(* IEC 61131-3 sources: std_i2980_v2.06_cp053/Source/IMM/ieccontrol/ODC1 (part 8) *)

(* ---- ABODC.pu ---- *)
(*
@h    ! WARNING !
@h    The Kemro K2 system (including software) only meets category B according to EN 954-1,
@h    thus it is not intended for usage in safety-relevant control applications in the field
@h    of personal safety (e.g. emergency stop).
@h    To implement potentially necessary safety-relevant control tasks, always use additional
@h    external safety devices that are intended for the particular purpose, and meet the necessary
@h    functional safety.
@h    For further information see EN 954-1 (EN ISO 13849-1) and/or the K2-x00 user manual, chapter
@h    "CE conformity, directives and standards".

*)

IMPORT_OVER_LISTFILE
 SET_ALARM
, START_PROCESS_ALGORITHM
, CHECK_REF
, STOP_PROCESS_ALGORITHM
, FCreateODCVersion
, SET_EVENT
, FGetCatConfigValueString
, cMinMoveIdent
, cCompMold
, cCompEjector
, cMoveBeginSequence
, cMoveEndSequence
, cCompInjection
, cMoveFwd
, cMoveBwd
, cMoveStartParallel
, cMoveEndParallel
, cMoveCooling
, cMoveShake
, cMoveOut
, cMoveNone
, cODCDependencyDontCare
, cCompCore
, cMoveFwdInterPos
, cMaxDeviceMovements
, cMaxODCSteps
, cCompNone
, cMovePlast
, cTimeOutSempahore
, cMaxStartConditions
, cCompOperationMode
, cMoveIncreaseShotCounter
, cMaxMoveDevicesRegistered
, cCycleTimeArraySize
, cAllDevIndex
, cMoveStartCondition
, cMinCompId
, ABInterpreter
, KODC_Builder
, FBGetMoveNumber
, FBAutoManual
, FBDebugTrace
, tsGlbSafetyData
, FBDebugTrace2
, KRTOS_Semaphore
, KODC_Sequence
, tyODCSequenceInternal
, KODC_Movements
, tnOperationMode
, tsStartedMoveDataODCExtended
, tyMovementRegisterList
, tsStartedMoveData
, tsODCDeviceMovementList
, tyODCSequenceBackup
, tnDataState
, tevStopRequest
, tevStartedStopped
, tevStartRequest
, ALARM_EVENT
, tsStartedMoveInfo
, tnODCRecalcMode
, KRTOS_Status
, tyStartCondInstanceData
, tevCheckLocklist
, tsTraceLevel
, tyStartConditionPosArray
, tsDeviceId
, tsActiveSequence
, tyLoopData
, tyODCParallelInfo
, tyStepBwdMovements
, tsSequenceDimension
, tevModifyCycleStartCondition
, tevCycleStart
, tyCycleTime
, ABSequDependencies
, RTC
, KODC_Step
, FBLockUnlock
, FBSetStepState
, tsODCStepPos
, ABODCCheckDependencies
, tMoveIdent
, FBStart
, tevCheckLocklistData
, tevStartRequestData
, tevStopRequestData
, FBStop
, FBCheckPosReached
, tevStartedStoppedData
, tsStartedMoveInfoODCExtended
, ABWaitCycleStart
, KSWO_Status
, ALARM_EVENT_DATA
, tyODCDependencyArray
, TON
, tevModifyCycleStartCondData
, FBAddDependency

END_IMPORT

ALGORITHM_BLOCK ABODC #DUMMY_EDIT_BLOCK

SYSTEM_VAR
 sv_ODCSequence : KODC_Sequence;
 sv_ODCSequenceInt : tyODCSequenceInternal;
 sv_ODCMovements : KODC_Movements;
 sv_dCycleDelaySet : TIME;
 sv_dCycleDelayAct : TIME;
 sv_bFirstCycle : BOOL;
 sv_bInitDone : BOOL;
 sv_bCombinedMovementsInManual : BOOL;
 sv_OperationMode : tnOperationMode;
 sv_StartedManualMovements : tsStartedMoveDataODCExtended;
 sv_MovementsAvailable : tyMovementRegisterList;
 sv_bODCFilesChanged : BOOL;
 sv_bProgramSwitchChanged : BOOL;
 sv_bActivationChanged : BOOL;
 sv_StartedMovements : tsStartedMoveData;
 sv_ODCDeviceMovements : tsODCDeviceMovementList (* list of all devices that registered movements for the ODC *);
 sv_iMovementsAvailable : DINT;
 sv_bAutoCycleRunning : BOOL;
 sv_dMaxCycleTime : TIME;
 sv_dCycleTime : TIME;
 sv_dCycleTimeMachine : TIME (* act. cylce time machine *);
 sv_ODCSequenceGenerateTime : DATE_AND_TIME;
 sv_ODCSequenceBackup : tyODCSequenceBackup;
 sv_iODCSequenceAct : DINT;
 sv_iSequenceToRestore : DINT;
 sv_ODCDescriptionPath : STRING(255);
 sv_DataState : tnDataState;
 sv_iODCSequenceUpdated : DINT;
 sv_iUsedRows : DINT;
 sv_iUsedColumns : DINT;
 sv_iInitOK : DINT (* 0 nothing initialized, 10 sequence array initialized, 20 sequence array + safety initialized *);
 sv_iActiveEditors : DINT;
 sv_StartConditionInstanceData : tyStartCondInstanceData (* list with start condition params for all instances *);
 sv_bUseProgramSwitches : BOOL (* TRUE: create sequence by using program switches; FALSE: use sequence from ODC editor *);
 sv_TraceLevel : tsTraceLevel;
 sv_dCalculatedCycleTime : TIME (* calculated cycle time (written by machine sequencer) *);
 sv_iEditorPropertiesChanged : DINT;
 sv_dAllowedCycleDeviation : TIME;
 sv_dLastCycleTime : TIME;
 sv_bTRUE : BOOL;
 sv_bODCCombinedMoveActive : BOOL (* TRUE: combined movement (for example closing sequence) is active (only in manual mode!) *);
 sv_DeviceId : tsDeviceId;
 sv_bOverrideCoreSafety : BOOL;
 sv_bOverrideEjectorSafety : BOOL;
 sv_ActiveSequence : tsActiveSequence;
 sv_LoopParameter : tyLoopData (* array with data of all programmed loops *);
 sv_InterpreterParallelInfo : tyODCParallelInfo (* internal state information of the interpreter, useful for HMI *);
 sv_bSequenceInterruption : BOOL (* TRUE: sequence is interrupted *);
 di_StepFwd : BOOL;
 di_StepBwd : BOOL;
 sv_bStepBwdActive : BOOL (* TRUE: stepping bwd is active *);
 sv_SequenceDimension : tsSequenceDimension (* contains the maximum size of the sequence array *);
 sv_bRecalcPendingOrActive : BOOL (* The ODC wants to recalc the sequence or a recalc is currently active. Any evStartRequest sent at this time can potentially be ignored if recalculation is already active. *);
END_VAR

SYSTEM_OBJECT
 evStopRequest : tevStopRequest;
 evStartedStopped : tevStartedStopped;
 evStartRequest : tevStartRequest;
 evAlarmFinishCycleAndStop : ALARM_EVENT;
 erODCInitFailed : ALARM;
 erCycleTimeExceeded : ALARM;
 EV_Task_3 : TASK;
 EV_Task_7 : TASK;
 PU_Task_3 : TASK;
 PU_Task_7 : TASK;
 TaskAnalog : TASK;
 TaskMid : TASK;
 erAssert : ALARM;
 TaskSlow : TASK;
 erCompNotInCorrectPosition : ALARM;
 erTeachModeActive : ALARM;
 evCheckLocklist : tevCheckLocklist;
 TaskSequencer : TASK;
 erMovementDuringActiveSequence : ALARM;
 erSequenceDuringActiveMovement : ALARM;
 erMachineSequenceNotCreated : ALARM;
 PU_Task_13 : TASK;
 erNoInverseMovement : ALARM;
 erTooManyStartParallel : ALARM;
 TaskInject : TASK;
 evModifyCycleStartCondition : tevModifyCycleStartCondition;
 evNewCycleStarted : tevCycleStart;
END_OBJECT

VAR_GLOBAL
 MovementsSema : KRTOS_Semaphore (* protects sv_StartedManualMovements *);
END_VAR

VAR_EXTERNAL
 g_SafetyData : tsGlbSafetyData;
 g_iAutoCycleLoopStartLine : DINT;
 g_iAutoCycleLoopEndLine : DINT;
 g_iODCMoveDevicesRegistered : DINT (* number of registered devices with ODC movements  *);
END_VAR

VAR
 abInterpreter : ABInterpreter;
 abKODC_Builder : KODC_Builder;
 fbGetMoveNumber : FBGetMoveNumber;
 fbAutoManual : FBAutoManual;
 fbDebugTrace : FBDebugTrace;
 fbDebugTrace2 : FBDebugTrace2;
 dummy : DINT;
 dummy2 : BOOL;
 mStartedCombinedMovement : tsStartedMoveInfo;
 mRecalcMode : tnODCRecalcMode (* currently active recalc mode, set by aDoPendingRecalc when the ODC decided to start recalculation of the sequence *);
 Status : KRTOS_Status;
 mbStopCycle : BOOL;
 mbStopAfterCycle : BOOL;
 mbCycleTimeRunning : BOOL;
 mbCycleTimeMachineRunning : BOOL (* condition for cycle time machine *);
 mbSequenceChanged : BOOL (* the ODC sequence array possibly changed->need to backup when first started *);
 mbIgnoreProgramSwitchChange : BOOL (* ignore program switch or activation changes during mold data loading *);
 mPendingRecalc : tnODCRecalcMode (* recalculations requested by aSetPendingRecalc but not started yet *);
 mbRecalcActive : BOOL;
 mbEjeBwdAtCycleStart : BOOL (* info if ejector must be bwd at the beginning of the cycle (taken from safety array of first step) *);
 miIndexEjectorInSafetyArray : DINT;
 mStartConditionPosArray : tyStartConditionPosArray (* array with information about the position of each start condition in the internal sequence *);
 mActiveStepBwdMovements : tyStepBwdMovements (* ArrayIndex = column number! *);
 mbResetCycleTime : BOOL;
 mbResetCycleTimeMachine : BOOL;
END_VAR

ALGORITHM aIsAnyColumnActive

VAR_OUTPUT
 bActive : BOOL;
END_VAR

VAR_TEMP
 i : DINT;
END_VAR
#BEGIN_EDIT_BLOCK
(**************************************** WARNING ********************************************
 *** The KEBA Kemro K2 System including software is not intended for safety control tasks! ***
 ***                       For further information see Comment tab!                        ***
 *********************************************************************************************)

bActive := FALSE;
FOR i := 2 TO sv_iUsedColumns DO
   IF sv_InterpreterParallelInfo[i].bColumnActive THEN
      bActive := TRUE;
      EXIT;
   END_IF;
END_FOR;

;#END_EDIT_BLOCK END_ALGORITHM

ALGORITHM aCheckCycleTime

VAR
 CycleTimeArray : tyCycleTime;
 i : DINT := 1;
 dSum : TIME;
 dAverageCycleTime : TIME;
END_VAR
#BEGIN_EDIT_BLOCK
(**************************************** WARNING ********************************************
 *** The KEBA Kemro K2 System including software is not intended for safety control tasks! ***
 ***                       For further information see Comment tab!                        ***
 *********************************************************************************************)

CycleTimeArray[i] := sv_dCycleTime;
dSum := dSum + CycleTimeArray[i];
i := i + 1;

IF i > cCycleTimeArraySize THEN
   //check if cycletime of last x - cycles is stable
   dAverageCycleTime := dSum / cCycleTimeArraySize;

   //-> check deviation between average cycle time and calculated cycle time
   IF (SUB_TIME(dAverageCycleTime, sv_dCalculatedCycleTime)) > sv_dAllowedCycleDeviation THEN
      sv_iEditorPropertiesChanged := sv_iEditorPropertiesChanged + 1;
   END_IF;

   i := 1;
   dSum := t#0s;
END_IF;

;#END_EDIT_BLOCK END_ALGORITHM

(*
Back up the current sequence (sv_ODCSequence)
A backup is only written when sv_ODCSequence is not equal to the last backup
*)

PROCESS_ALGORITHM paBackupSequence ON TaskSlow

#BEGIN_EDIT_BLOCK
(**************************************** WARNING ********************************************
 *** The KEBA Kemro K2 System including software is not intended for safety control tasks! ***
 ***                       For further information see Comment tab!                        ***
 *********************************************************************************************)

IF NOT mbSequenceChanged THEN
   fbDebugTrace2(nODCInterpreter, 'no sequence backup written as sequence did NOT change');
   STOP_PROCESS_ALGORITHM();
   RETURN;
END_IF;

mbSequenceChanged := FALSE;

IF sv_ODCSequenceBackup[sv_iODCSequenceAct].Sequence = sv_ODCSequence THEN
   fbDebugTrace2(nODCInterpreter, 'ODC sequences equal, doing nothing');
   STOP_PROCESS_ALGORITHM();
   RETURN;
END_IF;
fbDebugTrace2(nODCInterpreter, 'ODC sequences different, making backup');

sv_iODCSequenceAct := sv_iODCSequenceAct + 1;
IF sv_iODCSequenceAct > cODCSequenceBackupCount THEN
   sv_iODCSequenceAct := 1;
END_IF;

//FIXME: maybe do in smaller steps to avoid blocking the system for a long time
fbDebugTrace2(nODCInterpreter, CONCAT('saving new ODC sequence in history at pos ', DINT_TO_STRING(sv_iODCSequenceAct)));

sv_ODCSequenceBackup[sv_iODCSequenceAct].Sequence := sv_ODCSequence;
sv_ODCSequenceBackup[sv_iODCSequenceAct].Date := sv_ODCSequenceGenerateTime;
fbDebugTrace2(nODCInterpreter, 'saving backup done');

STOP_PROCESS_ALGORITHM();

;#END_EDIT_BLOCK END_ALGORITHM

(*
Queue a recalculation of the ODC sequence

nODCRecalcReloadFiles reload the ODC files from the CF + nODCRecalcCylce
nODCRecalcCylce       recalculate the cycle(because a program switch changed) + nODCRecalcSafety
nODCRecalcSafety      recalculate safety only(a movement was disabled)
*)

ALGORITHM aSetPendingRecalc

VAR_INPUT
 RecalcMode : tnODCRecalcMode (* How much of the ODC array to recalculate *);
END_VAR
#BEGIN_EDIT_BLOCK
(**************************************** WARNING ********************************************
 *** The KEBA Kemro K2 System including software is not intended for safety control tasks! ***
 ***                       For further information see Comment tab!                        ***
 *********************************************************************************************)

IF RecalcMode > mPendingRecalc THEN
   mPendingRecalc := RecalcMode;
   sv_bRecalcPendingOrActive := TRUE;
END_IF;

;#END_EDIT_BLOCK END_ALGORITHM

(*
Start a pending recalculation of the ODC sequence

If bStartedRecalc is TRUE then a pending recalculation was started.

To find out when recalculation finishes wait until mbRecalcActive is FALSE again
*)

ALGORITHM aDoPendingRecalc

VAR_OUTPUT
 bStartedRecalc : BOOL;
END_VAR
#BEGIN_EDIT_BLOCK
(**************************************** WARNING ********************************************
 *** The KEBA Kemro K2 System including software is not intended for safety control tasks! ***
 ***                       For further information see Comment tab!                        ***
 *********************************************************************************************)

bStartedRecalc := FALSE;

IF mPendingRecalc = nODCRecalcNone THEN
   RETURN;
END_IF;

IF mbRecalcActive THEN
   fbDebugTrace('another ODC recalc is already active, new recalc will be executed later');
   RETURN;
END_IF;

IF mPendingRecalc > mRecalcMode THEN
   mRecalcMode := mPendingRecalc;
END_IF;
// mRecalcMode will be reset after the recalc finished successfully
// but keeps the value if an error occured
// this way we can be sure the right recalc mode is used when
// the first recalc with nODCRecalcCylce fails and the second recalc with only nODCRecalcSafety succeeds
// the cycle is recalculated, and not only safety

mPendingRecalc := nODCRecalcNone;

IF mRecalcMode = nODCRecalcReloadFiles THEN
   fbDebugTrace2(nODCInterpreter, 'start initializing ODC array WITH reading new files');
ELSIF mRecalcMode = nODCRecalcCylce THEN
   fbDebugTrace2(nODCInterpreter, 'start initializing ODC array WITHOUT reading new files');
ELSIF mRecalcMode = nODCRecalcSafety THEN
   fbDebugTrace2(nODCInterpreter, 'start initializing ODC dependency array');
ELSIF mRecalcMode = nODCRecalcInternal THEN
   fbDebugTrace2(nODCInterpreter, 'start initializing internal ODC array');
ELSE
   fbDebugTrace2(nODCInterpreter, 'NOT starting initialization of ODC because we got a strange reason');
   RETURN;
END_IF;

bStartedRecalc := TRUE;
mbRecalcActive := TRUE; //set flag immediately, do not wait for PA, which might be delayed a bit because it is low prio
START_PROCESS_ALGORITHM(paInitSequence);

;#END_EDIT_BLOCK END_ALGORITHM

(*
Does the (re)initialisation of the ODC sequence and saves
the sequence generation time

*)

PROCESS_ALGORITHM paInitSequence ON TaskMid

VAR_TEMP
 iTmpRow : DINT;
 iTmpCol : DINT;
 iMove : DINT;
 iDevice : DINT;
 k : DINT;
 i : DINT;
 iTmpCol2 : DINT (* column *);
 iTmpRow2 : DINT (* line *);
END_VAR

VAR
 iCalledInit : DINT;
 iCalledCreate : DINT;
 bInitDone : BOOL;
 abSequDependencies : ABSequDependencies;
 fbRTC : RTC;
 bError : BOOL;
 RecalcMode : tnODCRecalcMode;
 sPath : STRING(255);
 bFirstCall : BOOL;
 sWorkPath : STRING(255);
 iInstance : DINT;
 fbLockUnlockAll : FBLockUnlock := (DeviceId:=(CompId:=cCompAll,IndexId:=cAllDevIndex),MoveDir:=cMoveAll,MoveId:=cMoveAll);
 DeviceId : tsDeviceId;
 bTryAgain : BOOL;
 FailedRecalc : tnODCRecalcMode;
 iCount : INT;
 iOrigEndLine : DINT;
 StepBeginLoop : KODC_Step := (iCompId:=cCompODC,iMoveDir:=cMoveNone,iMoveId:=cMoveBeginLoop,iIndexId:=1,iCount:=1);
 StepEndLoop : KODC_Step := (iCompId:=cCompODC,iMoveDir:=cMoveNone,iMoveId:=cMoveEndLoop,iIndexId:=1,iCount:=1);
 bAddLoop : BOOL;
 iTmp : DINT;
 DeviceIdEjector1 : tsDeviceId := (CompId:=cCompEjector,IndexId:=1);
 DependencyEjectorBwd : LWORD (* dependency which represents "ejector bwd" *);
 bInit : BOOL;
 iNoOfStartParallel : DINT;
END_VAR

VAR CONSTANT
 EmptySequenceEntry : KODC_Step := (iCompId:=cCompNone,iMoveDir:=cMoveNone,iMoveId:=cMoveNone,iIndexId:=1,iCount:=0);
END_VAR

(* IecGraph-Code *)

(* init step *)
INITIAL_STEP SStart:
AStart (P);
AInitAdditionalMoveData (P);
AResetProgrammedInSequence (P);
END_STEP

ACTION AStart: #BEGIN_EDIT_BLOCK
fbDebugTrace2(nODCInterpreter, 'starting initialisation of ODC sequence');

RESET_ALARM(Name := erODCInitFailed);

RecalcMode := mRecalcMode;
FailedRecalc := mRecalcMode;  //remember in case of failed recalc so we can repeat
mRecalcMode := nODCRecalcNone;

sv_iInitOK := 0;

(* lock all movements so nothing can happen during init *)
fbLockUnlockAll.Alarm.AlarmId := erMachineSequenceNotCreated;
fbLockUnlockAll(Mode := nLockAbort);

;#END_EDIT_BLOCK END_ACTION (*AStart*)

(* steps *)
STEP SError:
AError (N);
END_STEP

ACTION AError: #BEGIN_EDIT_BLOCK
fbDebugTrace('initializing ODC array NOT successful');

(* set the generic erODCInitFailed ALARM which will block machine operation
   for detailed information other alarms are set which explain 1 or more problems
   of the ODC sequence *)
SET_ALARM(Name := erODCInitFailed);

mbRecalcActive := FALSE;

//reset mRecalcMode
//this way a failed recalc can not be replaced by a succeeding recalc
//of lower priority
mRecalcMode := FailedRecalc;

// indicate an update of the odc list so the hmi can react properly
sv_iODCSequenceUpdated := sv_iODCSequenceUpdated + 1;

//notify other code parts when recalc is finished (in this case unsuccessfully)
sv_bRecalcPendingOrActive := FALSE;

STOP_PROCESS_ALGORITHM();

;#END_EDIT_BLOCK END_ACTION (*AError*)
STEP Step28:
END_STEP

STEP SInitSequence:
AInit1 (P);
AInit2 (N);
END_STEP

ACTION AInit1: #BEGIN_EDIT_BLOCK
iCalledInit := 0;
iCalledCreate := 0;

IF NOT bFirstCall THEN
   sWorkPath := FGetCatConfigValueString('System.workPath', '/harddisk0/');
   bFirstCall := TRUE;
END_IF;

sPath := CONCAT(sWorkPath, sv_ODCDescriptionPath);
abKODC_Builder.Init(Movements := sv_ODCMovements, DescriptionFilePath := sPath, Execute := FALSE);

;#END_EDIT_BLOCK END_ACTION (*AInit1*)
ACTION AInit2: #BEGIN_EDIT_BLOCK
abKODC_Builder.Init(Execute := TRUE);
iCalledInit := iCalledInit + 1;

;#END_EDIT_BLOCK END_ACTION (*AInit2*)
STEP SInitSequenceDone:
AInit3 (P);
END_STEP

ACTION AInit3: #BEGIN_EDIT_BLOCK
IF abKODC_Builder.Init.Error AND abKODC_Builder.Init.Done THEN
   fbDebugTrace2(nODCInterpreter, 'ERROR init returned success and failure at the same time');
END_IF;

IF abKODC_Builder.Init.Done THEN
   fbDebugTrace2(nODCInterpreter, CONCAT('called init ',
                                         DINT_TO_STRING(iCalledInit),
                                         ' times then it returned success'));
ELSIF abKODC_Builder.Init.Error THEN
   fbDebugTrace2(nODCInterpreter, CONCAT('called init ',
                                         DINT_TO_STRING(iCalledInit),
                                         ' times then it returned error'));
END_IF;

;#END_EDIT_BLOCK END_ACTION (*AInit3*)
STEP Step16:
END_STEP

STEP SCreateSequence:
AClearSequence (P);
ACreateSequence1 (P);
ACreateSequence2 (N);
END_STEP

ACTION ACreateSequence1: #BEGIN_EDIT_BLOCK
fbDebugTrace2(nODCInterpreter, 'initialisation of ODC array');
(* WARNING: Columns and Rows must be <= the real size of the array
   otherwise the builder will write outside of the array
   and memory corruption will occur ! *)
abKODC_Builder.CreateSequence(Sequence := sv_ODCSequence, Columns := cMaxParallelMovements, Rows := cMaxODCSteps, Execute := FALSE);

;#END_EDIT_BLOCK END_ACTION (*ACreateSequence1*)
ACTION ACreateSequence2: #BEGIN_EDIT_BLOCK
abKODC_Builder.CreateSequence(Execute := TRUE);
iCalledCreate := iCalledCreate + 1;

;#END_EDIT_BLOCK END_ACTION (*ACreateSequence2*)
STEP SCreateSequenceDone:
ACreateSequence3 (P);
END_STEP

ACTION ACreateSequence3: #BEGIN_EDIT_BLOCK
IF abKODC_Builder.CreateSequence.Error AND abKODC_Builder.CreateSequence.Done THEN
   fbDebugTrace2(nODCInterpreter, 'ERROR CreateSequence returned success and failure at the same time');
END_IF;

IF abKODC_Builder.CreateSequence.Done THEN
   fbDebugTrace2(nODCInterpreter, CONCAT('called CreateSequence ',
                                         DINT_TO_STRING(iCalledCreate),
                                         ' times then it returned success'));
ELSIF abKODC_Builder.CreateSequence.Error THEN
   fbDebugTrace2(nODCInterpreter, CONCAT('called CreateSequence ',
                                         DINT_TO_STRING(iCalledCreate),
                                         ' times then it returned error'));
END_IF;

;#END_EDIT_BLOCK END_ACTION (*ACreateSequence3*)
STEP SSanityCheckAndNumber:
ACheckSequenceDimension (P);
AInitEmptySteps (P);
ASanity (P);
END_STEP

ACTION ASanity: #BEGIN_EDIT_BLOCK
bError := FALSE;
abInterpreter.aCheckSequenceSanity();
IF NOT abInterpreter.aCheckSequenceSanity.bOK THEN
   fbDebugTrace('checking sanity of ODC array failed');
   bError := TRUE;
   RETURN;
END_IF;
bAddLoop := NOT abInterpreter.aCheckSequenceSanity.bAutoCycleLoopFound;
iNoOfStartParallel := abInterpreter.aCheckSequenceSanity.iNoOfStartParallel;

;#END_EDIT_BLOCK END_ACTION (*ASanity*)
STEP Step33:
END_STEP

STEP S_AddCycleLoop:
AInsertAutoCycleLoop (P);
END_STEP

STEP Step32:
ACreateInternalSequence (P);
END_STEP

ACTION ACreateInternalSequence: #BEGIN_EDIT_BLOCK
bError := FALSE;
abInterpreter.aClearInternalSequence();

abInterpreter.aCreateInternalSequence();
IF abInterpreter.aCreateInternalSequence.bError THEN
   fbDebugTrace('aCreateInternalSequence failed');
   bError := TRUE;
   RETURN;
END_IF;

sv_iUsedColumns := abInterpreter.aCreateInternalSequence.iUsedColumns;
sv_iUsedRows := abInterpreter.aCreateInternalSequence.iUsedRows;

// save sequence generation time
fbRTC(EN := FALSE);
sv_ODCSequenceGenerateTime := fbRTC.CDT;
mbSequenceChanged := TRUE;

;#END_EDIT_BLOCK END_ACTION (*ACreateInternalSequence*)
STEP Step26:
AInitSequenceOK (N);
END_STEP

ACTION AInitSequenceOK: #BEGIN_EDIT_BLOCK
sv_iInitOK := 10;

;#END_EDIT_BLOCK END_ACTION (*AInitSequenceOK*)
STEP SBeforeRecalcSafety:
END_STEP

STEP SRecalcSafety:
ACalcSeqDependencies (P);
ASetProgrammedInSequence (P);
END_STEP

ACTION ACalcSeqDependencies: #BEGIN_EDIT_BLOCK
IF iNoOfStartParallel <= cMaxStartParallel THEN
   RESET_ALARM(Name := erTooManyStartParallel);
   abSequDependencies.aCalc();
   IF abSequDependencies.aCalc.bError THEN
      bError := TRUE;
      fbDebugTrace('sequence dependency calculation returned a error');
   END_IF;
ELSE
   SET_ALARM(Name := erTooManyStartParallel);
END_IF;

;#END_EDIT_BLOCK END_ACTION (*ACalcSeqDependencies*)
STEP S_Check_Pending_Recalc:
ACheckForPendingRecalc (P);
END_STEP

ACTION ACheckForPendingRecalc: #BEGIN_EDIT_BLOCK
bTryAgain := FALSE;
IF mPendingRecalc <> nODCRecalcNone THEN
   //recalc during creation of sequence requested
   //=> ignore result and start again
   mRecalcMode := mPendingRecalc;
   mPendingRecalc := nODCRecalcNone;
   bTryAgain := TRUE;
END_IF;

;#END_EDIT_BLOCK END_ACTION (*ACheckForPendingRecalc*)
STEP SFinish:
ACheckEjeBwdAtCycleStart (P);
AFinish (N);
END_STEP

ACTION AFinish: #BEGIN_EDIT_BLOCK
(* array ok -> unlock all movements *)
fbLockUnlockAll.Alarm.AlarmId := erMachineSequenceNotCreated;
fbLockUnlockAll(Mode := nUnlock);

abInterpreter.aSetInitOK();
fbDebugTrace2(nODCInterpreter, 'initializing ODC array successful');

mbRecalcActive := FALSE;

// indicate an update of the odc list so the hmi can react properly
sv_iInitOK := 20;
sv_iODCSequenceUpdated := sv_iODCSequenceUpdated + 1;

//notify other code parts when recalc is finished (and it is OK to send an evStartRequest)
sv_bRecalcPendingOrActive := FALSE;

STOP_PROCESS_ALGORITHM();

;#END_EDIT_BLOCK END_ACTION (*AFinish*)

(* transitions *)
TRANSITION Trans25 (* Trans25 *) FROM SError TO SStart :=  #BEGIN_EDIT_BLOCK
TRUE
;#END_EDIT_BLOCK
END_TRANSITION

GO_ON_TRANSITION Trans38 (* Trans38 *) FROM SStart TO Step28 :=  #BEGIN_EDIT_BLOCK
RecalcMode <> nODCRecalcInternal
;#END_EDIT_BLOCK
END_TRANSITION

GO_ON_TRANSITION TNewSequenceFromEditor (* Trans39 *) FROM SStart TO SSanityCheckAndNumber :=  #BEGIN_EDIT_BLOCK
RecalcMode = nODCRecalcInternal
;#END_EDIT_BLOCK
END_TRANSITION

GO_ON_TRANSITION Trans13 (* Trans13 *) FROM Step28 TO Step16 :=  #BEGIN_EDIT_BLOCK
NOT (RecalcMode >= nODCRecalcReloadFiles)
;#END_EDIT_BLOCK
END_TRANSITION

GO_ON_TRANSITION TRecalcReloadFiles (* Trans12 *) FROM Step28 TO SInitSequence :=  #BEGIN_EDIT_BLOCK
RecalcMode >= nODCRecalcReloadFiles
;#END_EDIT_BLOCK
END_TRANSITION

TRANSITION Trans2 (* Trans2 *) FROM SInitSequence TO SInitSequenceDone :=  #BEGIN_EDIT_BLOCK
abKODC_Builder.Init.Done OR abKODC_Builder.Init.Error
;#END_EDIT_BLOCK
END_TRANSITION

GO_ON_TRANSITION Trans11 (* Trans11 *) FROM SInitSequenceDone TO Step16 :=  #BEGIN_EDIT_BLOCK
NOT abKODC_Builder.Init.Error
;#END_EDIT_BLOCK
END_TRANSITION

GO_ON_TRANSITION Trans26 (* Trans26 *) FROM SInitSequenceDone TO SError :=  #BEGIN_EDIT_BLOCK
abKODC_Builder.Init.Error
;#END_EDIT_BLOCK
END_TRANSITION

GO_ON_TRANSITION Trans20 (* Trans20 *) FROM Step16 TO SBeforeRecalcSafety :=  #BEGIN_EDIT_BLOCK
NOT (RecalcMode >= nODCRecalcCylce)
;#END_EDIT_BLOCK
END_TRANSITION

GO_ON_TRANSITION TRecalcCycle (* Trans19 *) FROM Step16 TO SCreateSequence :=  #BEGIN_EDIT_BLOCK
RecalcMode >= nODCRecalcCylce
;#END_EDIT_BLOCK
END_TRANSITION

TRANSITION Trans4 (* Trans4 *) FROM SCreateSequence TO SCreateSequenceDone :=  #BEGIN_EDIT_BLOCK
abKODC_Builder.CreateSequence.Error OR abKODC_Builder.CreateSequence.Done
;#END_EDIT_BLOCK
END_TRANSITION

GO_ON_TRANSITION Trans27 (* Trans27 *) FROM SCreateSequenceDone TO SSanityCheckAndNumber :=  #BEGIN_EDIT_BLOCK
NOT abKODC_Builder.CreateSequence.Error
;#END_EDIT_BLOCK
END_TRANSITION

GO_ON_TRANSITION Trans28 (* Trans28 *) FROM SCreateSequenceDone TO SError :=  #BEGIN_EDIT_BLOCK
abKODC_Builder.CreateSequence.Error
;#END_EDIT_BLOCK
END_TRANSITION

GO_ON_TRANSITION Trans46 (* Trans46 *) FROM SSanityCheckAndNumber TO Step33 :=  #BEGIN_EDIT_BLOCK
NOT bError
;#END_EDIT_BLOCK
END_TRANSITION

GO_ON_TRANSITION Trans50 (* Trans50 *) FROM SSanityCheckAndNumber TO SError :=  #BEGIN_EDIT_BLOCK
bError
;#END_EDIT_BLOCK
END_TRANSITION

GO_ON_TRANSITION Trans48 (* Trans48 *) FROM Step33 TO S_AddCycleLoop :=  #BEGIN_EDIT_BLOCK
bAddLoop
;#END_EDIT_BLOCK
END_TRANSITION

TRANSITION TLoopAdded (* Trans50 *) FROM S_AddCycleLoop TO Step32 :=  #BEGIN_EDIT_BLOCK
TRUE
;#END_EDIT_BLOCK
END_TRANSITION

GO_ON_TRANSITION Trans49 (* Trans49 *) FROM Step33 TO Step32 :=  #BEGIN_EDIT_BLOCK
NOT bAddLoop
;#END_EDIT_BLOCK
END_TRANSITION

TRANSITION Trans14 (* Trans14 *) FROM Step32 TO Step26 :=  #BEGIN_EDIT_BLOCK
NOT bError
;#END_EDIT_BLOCK
END_TRANSITION

GO_ON_TRANSITION Trans36 (* Trans36 *) FROM Step26 TO SBeforeRecalcSafety :=  #BEGIN_EDIT_BLOCK
TRUE
;#END_EDIT_BLOCK
END_TRANSITION

TRANSITION Trans29 (* Trans29 *) FROM Step32 TO SError :=  #BEGIN_EDIT_BLOCK
bError
;#END_EDIT_BLOCK
END_TRANSITION

GO_ON_TRANSITION Trans22 (* Trans22 *) FROM SBeforeRecalcSafety TO S_Check_Pending_Recalc :=  #BEGIN_EDIT_BLOCK
NOT (RecalcMode >= nODCRecalcSafety)
;#END_EDIT_BLOCK
END_TRANSITION

GO_ON_TRANSITION TRecalcSafety (* Trans23 *) FROM SBeforeRecalcSafety TO SRecalcSafety :=  #BEGIN_EDIT_BLOCK
RecalcMode >= nODCRecalcSafety
;#END_EDIT_BLOCK
END_TRANSITION

GO_ON_TRANSITION Trans24 (* Trans24 *) FROM SRecalcSafety TO S_Check_Pending_Recalc :=  #BEGIN_EDIT_BLOCK
NOT bError
;#END_EDIT_BLOCK
END_TRANSITION

GO_ON_TRANSITION Trans30 (* Trans30 *) FROM SRecalcSafety TO SError :=  #BEGIN_EDIT_BLOCK
bError
;#END_EDIT_BLOCK
END_TRANSITION

GO_ON_TRANSITION TNoRecalc (* Trans44 *) FROM S_Check_Pending_Recalc TO SFinish :=  #BEGIN_EDIT_BLOCK
NOT bTryAgain
;#END_EDIT_BLOCK
END_TRANSITION

GO_ON_TRANSITION TRecalc (* Trans45 *) FROM S_Check_Pending_Recalc TO SStart :=  #BEGIN_EDIT_BLOCK
bTryAgain
;#END_EDIT_BLOCK
END_TRANSITION

TRANSITION Trans8 (* Trans8 *) FROM SFinish TO SStart :=  #BEGIN_EDIT_BLOCK
TRUE
;#END_EDIT_BLOCK
END_TRANSITION

(* end IecGraph-Code *)
(* sfc-code *)

(* stand alone actions *)
ACTION AClearSequence: #BEGIN_EDIT_BLOCK
(* make sure the array is clean
   important for testing when 2 different partially initialized
   arrays are used *)
FOR iTmpCol := 1 TO cMaxParallelMovements DO
   FOR iTmpRow := 1 TO cMaxODCSteps DO
      sv_ODCSequence[iTmpCol][iTmpRow] := EmptySequenceEntry;
   END_FOR;
END_FOR;

;#END_EDIT_BLOCK END_ACTION (*AClearSequence*)
ACTION AInitAdditionalMoveData: #BEGIN_EDIT_BLOCK
(**************************************** WARNING ********************************************
 *** The KEBA Kemro K2 System including software is not intended for safety control tasks! ***
 ***                       For further information see Comment tab!                        ***
 *********************************************************************************************)
IF NOT bInitDone THEN

   //get FuIndex of all registered movements
   //fuIndex = index of the device in sv_ODCDeviceMovements
   FOR iMove := 1 TO sv_iMovementsAvailable DO
      FOR iDevice := 1 TO sv_ODCDeviceMovements.iCount DO
         IF sv_MovementsAvailable[iMove].DeviceId = sv_ODCDeviceMovements.Devices[iDevice].DeviceId THEN
            sv_MovementsAvailable[iMove].iFuIndex := iDevice;
            EXIT;
         END_IF;
      END_FOR;
   END_FOR;

   //get number of default movement for every device in sv_ODCDeviceMovements
   FOR iDevice := 1 TO sv_ODCDeviceMovements.iCount DO
      DeviceId := sv_ODCDeviceMovements.Devices[iDevice].DeviceId;
      FOR iMove := 1 TO sv_iMovementsAvailable DO
         IF sv_MovementsAvailable[iMove].DeviceId = DeviceId AND sv_MovementsAvailable[iMove].pMovementData^.bDefaultPos THEN
            //default movement found
            sv_ODCDeviceMovements.Devices[iDevice].iDefaultMoveNumber := iMove;
            EXIT;
         END_IF;
      END_FOR;
   END_FOR;

   bInitDone := TRUE;

END_IF;

;#END_EDIT_BLOCK END_ACTION (*AInitAdditionalMoveData*)
ACTION AResetProgrammedInSequence: #BEGIN_EDIT_BLOCK
(**************************************** WARNING ********************************************
 *** The KEBA Kemro K2 System including software is not intended for safety control tasks! ***
 ***                       For further information see Comment tab!                        ***
 *********************************************************************************************)

IF RecalcMode = nODCRecalcNone OR RecalcMode = nODCRecalcSafety THEN
   ;//no change in sequence
ELSE
   //sequence changed -> reset bProgrammedInSequence for all movements
   FOR iMove := 1 TO sv_iMovementsAvailable DO
      sv_MovementsAvailable[iMove].pMovementData^.bProgrammedInSequence := FALSE;

      IF sv_MovementsAvailable[iMove].pMovementData^.bInstanceable AND
        CHECK_REF(sv_MovementsAvailable[iMove].pMovementData^.InstanceData.pProgrammedInSequenceArray^) THEN

         //movement instanceable -> init programmed in sequence for all instances
         FOR k:= 1 TO cMaxIntermediateConditions DO
            sv_MovementsAvailable[iMove].pMovementData^.InstanceData.pProgrammedInSequenceArray^[k] := FALSE;
         END_FOR;

      END_IF;
   END_FOR;

   //reset array with start condition positions
   FOR i := 1 TO cMaxStartConditions DO
      mStartConditionPosArray[i].iColumn := 0;
      mStartConditionPosArray[i].iRow := 0;
   END_FOR;
END_IF;

;#END_EDIT_BLOCK END_ACTION (*AResetProgrammedInSequence*)
ACTION ASetProgrammedInSequence: #BEGIN_EDIT_BLOCK
(**************************************** WARNING ********************************************
 *** The KEBA Kemro K2 System including software is not intended for safety control tasks! ***
 ***                       For further information see Comment tab!                        ***
 *********************************************************************************************)

//set bProgrammedInSequence for all movements which are
//included in the created sequence
FOR iTmpRow := 1 TO sv_iUsedRows DO
   FOR iTmpCol := 1 TO sv_iUsedColumns DO
      iMove := sv_ODCSequenceInt[iTmpCol,iTmpRow].iMoveNumber;
      IF iMove >= cMoveNone THEN
         sv_MovementsAvailable[iMove].pMovementData^.bProgrammedInSequence := TRUE;

         IF sv_MovementsAvailable[iMove].pMovementData^.bInstanceable AND
           CHECK_REF(sv_MovementsAvailable[iMove].pMovementData^.InstanceData.pProgrammedInSequenceArray^) THEN
            //movement instanceable -> set programmed in sequence for according instance
            iInstance := sv_ODCSequenceInt[iTmpCol,iTmpRow].iCount;
            sv_MovementsAvailable[iMove].pMovementData^.InstanceData.pProgrammedInSequenceArray^[iInstance] := TRUE;
         END_IF;

      END_IF;

      //save position if step is a start condition
      IF sv_ODCSequence[iTmpCol,iTmpRow].iMoveId = cMoveStartCondition THEN
         iCount := sv_ODCSequence[iTmpCol, iTmpRow].iCount;
         mStartConditionPosArray[iCount].iColumn := iTmpCol;
         mStartConditionPosArray[iCount].iRow := iTmpRow;
      END_IF;

   END_FOR;
END_FOR;

;#END_EDIT_BLOCK END_ACTION (*ASetProgrammedInSequence*)
ACTION ACheckEjeBwdAtCycleStart: #BEGIN_EDIT_BLOCK
(**************************************** WARNING ********************************************
 *** The KEBA Kemro K2 System including software is not intended for safety control tasks! ***
 ***                       For further information see Comment tab!                        ***
 *********************************************************************************************)

//get index of ejector 1 in sv_ODCDeviceMovements
//and also get dependency which represents "Ejector bwd"
IF NOT bInit THEN
   FOR i := 1 TO g_iODCMoveDevicesRegistered DO
      IF sv_ODCDeviceMovements.Devices[i].DeviceId = DeviceIdEjector1 THEN
         miIndexEjectorInSafetyArray := i;

         //find ejector bwd movement
         FOR k := 1 TO sv_ODCDeviceMovements.Devices[miIndexEjectorInSafetyArray].iNumberOfMovements DO
            IF sv_ODCDeviceMovements.Devices[miIndexEjectorInSafetyArray].Movements[k]^.MoveId = cMoveBwd THEN

               //movement found in sv_ODCDeviceMovements -> set the according bit
               DependencyEjectorBwd := cFirstBit;

               //first movement: shift right 0, second movement: shift right 1, ...
               DependencyEjectorBwd := SHR(DependencyEjectorBwd, (k-1));
               EXIT;
            END_IF;
         END_FOR;

         EXIT;
      END_IF;
   END_FOR;
   bInit := TRUE;
END_IF;

//avoid problems if no ejector is available
mbEjeBwdAtCycleStart := FALSE;
IF miIndexEjectorInSafetyArray > 0 THEN
   //check dependency array of first step and find out if ejector must be bwd
   IF sv_ODCSequenceInt[1,1].SafetyArray[miIndexEjectorInSafetyArray].Dependency = DependencyEjectorBwd THEN
      mbEjeBwdAtCycleStart := TRUE;
   END_IF;
END_IF;

;#END_EDIT_BLOCK END_ACTION (*ACheckEjeBwdAtCycleStart*)
ACTION AInsertAutoCycleLoop: #BEGIN_EDIT_BLOCK
(**************************************** WARNING ********************************************
 *** The KEBA Kemro K2 System including software is not intended for safety control tasks! ***
 ***                       For further information see Comment tab!                        ***
 *********************************************************************************************)

IF sv_TraceLevel.bODCInterpreter THEN
   dummy := Print('No AutoCycleLoop found ----> add LOOP automatically');
END_IF;

iOrigEndLine := abInterpreter.aCheckSequenceSanity.iEndSequenceRow;
IF sv_TraceLevel.bODCInterpreter THEN
   dummy := Print('original end line: %d', iOrigEndLine);
END_IF;

//move line with ODC.EndSequence two lines down
//add ODC.EndLoop before ODC.EndSequence
//move the whole sequence one line down
//add ODC.BeginLoop in second line (first line is ODC.BeginSequence)
//fill sv_LoopData with correct values

FOR iTmpCol2 := 1 TO cMaxParallelMovements DO
   sv_ODCSequence[iTmpCol2,(iOrigEndLine+2)] := sv_ODCSequence[iTmpCol2, iOrigEndLine];
END_FOR;

IF sv_TraceLevel.bODCInterpreter THEN
   iTmp := iOrigEndLine +1;
   dummy := Print('Adding end loop in line %d', iTmp);
END_IF;

sv_ODCSequence[1,(iOrigEndLine+1)] := StepEndLoop;
g_iAutoCycleLoopEndLine := (iOrigEndLine+1);

FOR iTmpRow2 := iOrigEndLine TO 2 BY -1 DO
   FOR iTmpCol2 := 1 TO cMaxParallelMovements DO
      sv_ODCSequence[iTmpCol2,iTmpRow2] := sv_ODCSequence[iTmpCol2,(iTmpRow2-1)];
   END_FOR;
END_FOR;

IF sv_TraceLevel.bODCInterpreter THEN
   dummy := Print('Adding begin loop in line 2');
END_IF;
sv_ODCSequence[1,2] := StepBeginLoop;
g_iAutoCycleLoopStartLine := 2;

sv_LoopParameter[1].sTextKey := 'TxtAutoCycleLoop';
sv_LoopParameter[1].sVariable1 := 'system.sv_bFALSE';
sv_LoopParameter[1].sVariable2 := 'system.sv_bTRUE';
sv_LoopParameter[1].CompareOperator := nCompOperatorEqual;

;#END_EDIT_BLOCK END_ACTION (*AInsertAutoCycleLoop*)
ACTION AInitEmptySteps: #BEGIN_EDIT_BLOCK
(**************************************** WARNING ********************************************
 *** The KEBA Kemro K2 System including software is not intended for safety control tasks! ***
 ***                       For further information see Comment tab!                        ***
 *********************************************************************************************)

//performance optimization:
//at empty steps the machine sequencer only sets iCompId to cMinCompId
//iMoveId, iMoveDir, ... are not changed and keep the "old" values
//=> this steps must be set to "empty" steps in the IEC code
FOR iTmpCol := 1 TO cMaxParallelMovements DO
   FOR iTmpRow := 1 TO cMaxODCSteps DO
      IF (sv_ODCSequence[iTmpCol][iTmpRow].iCompId = cMinCompId) AND (sv_ODCSequence[iTmpCol][iTmpRow].iMoveId <> cMoveNone) THEN
         //set the whole step to "Empty"
         sv_ODCSequence[iTmpCol][iTmpRow] := EmptySequenceEntry;
      END_IF;
   END_FOR;
END_FOR;

;#END_EDIT_BLOCK END_ACTION (*AInitEmptySteps*)
ACTION ACheckSequenceDimension: #BEGIN_EDIT_BLOCK
(**************************************** WARNING ********************************************
 *** The KEBA Kemro K2 System including software is not intended for safety control tasks! ***
 ***                       For further information see Comment tab!                        ***
 *********************************************************************************************)

IF (sv_SequenceDimension.iMaxColumns > 0) AND (sv_SequenceDimension.iMaxRows > 0) THEN

   IF sv_SequenceDimension.iMaxColumns < cMaxParallelMovements THEN
      //loaded sequence is smaller (lower number of columns) than the actual sequence
      //-> init the rest of the columns
      FOR iTmpCol := (sv_SequenceDimension.iMaxColumns + 1) TO cMaxParallelMovements DO
         FOR iTmpRow := 1 TO cMaxODCSteps DO
            sv_ODCSequence[iTmpCol][iTmpRow] := EmptySequenceEntry;
         END_FOR;
      END_FOR;
   END_IF;

   IF sv_SequenceDimension.iMaxRows < cMaxODCSteps THEN
      //loaded sequence is smaller (lower number of rows) than the actual sequence
      //-> init the rest of the rows
      FOR iTmpCol := 1 TO sv_SequenceDimension.iMaxColumns DO
         FOR iTmpRow := (sv_SequenceDimension.iMaxRows + 1) TO cMaxODCSteps DO
            sv_ODCSequence[iTmpCol][iTmpRow] := EmptySequenceEntry;
         END_FOR;
      END_FOR;
   END_IF;
ELSE
   ;//loaded data does not contain the sequence dimension (=> data was created with a KePlast version < 01.38)
   //Attention:
   //It is not possible to automatically assume that the sequence dimension is 6 columns and 100 rows
   //in this case, because maybe in some customer projects the sequence size was already increased in
   //KePlast versions < 01.38
END_IF;

//set dimension to actual implemented array size
sv_SequenceDimension.iMaxColumns := cMaxParallelMovements;
sv_SequenceDimension.iMaxRows := cMaxODCSteps;

;#END_EDIT_BLOCK END_ACTION (*ACheckSequenceDimension*)
(* end sfc-code *)

END_ALGORITHM

ALGORITHM aClearStepState

VAR_INPUT
 bExcludeActiveColumns : BOOL;
END_VAR

VAR_TEMP
 iTmpRow : DINT;
 iTmpColumn : DINT;
END_VAR

VAR
 fbSetStepState : FBSetStepState;
END_VAR
#BEGIN_EDIT_BLOCK
(**************************************** WARNING ********************************************
 *** The KEBA Kemro K2 System including software is not intended for safety control tasks! ***
 ***                       For further information see Comment tab!                        ***
 *********************************************************************************************)

fbDebugTrace2(nODCInterpreter, 'begin clearing step state');

FOR iTmpRow := 1 TO sv_iUsedRows DO
   fbSetStepState.StepState := nStateDefault;
   fbSetStepState.StepPos.iRow := iTmpRow;

   FOR iTmpColumn := 1 TO sv_iUsedColumns DO
      fbSetStepState.StepPos.iColumn := iTmpColumn;

      IF NOT (bExcludeActiveColumns AND sv_InterpreterParallelInfo[iTmpColumn].bColumnActive) THEN
         //reset step state depending on bExcludeActiceColumns
         fbSetStepState();
      END_IF;

   END_FOR;
END_FOR;

fbDebugTrace2(nODCInterpreter, 'finished clearing step state');

;#END_EDIT_BLOCK END_ALGORITHM

(*
Start a single movement (in response to evStartRequest)
*)

ALGORITHM aStartAndCheckConditions

VAR_INPUT
 StepPos : tsODCStepPos;
 bNoAlarms : BOOL (* TRUE: alarms of not fulfilled conditions are not set *);
END_VAR

VAR_OUTPUT
 bCheckConditionsOk : BOOL;
 bStartConditionOk : BOOL;
 bCheckConditionFound : BOOL;
 iStartConditionsNotOk : DINT (* number of not fulfilled startconditions *);
 iCheckConditionsNotOk : DINT (* number of not fulfilled checkconditions *);
END_VAR

VAR_TEMP
 i : DINT;
END_VAR

VAR
 abODCCheckDependencies : ABODCCheckDependencies;
END_VAR
#BEGIN_EDIT_BLOCK
(**************************************** WARNING ********************************************
 *** The KEBA Kemro K2 System including software is not intended for safety control tasks! ***
 ***                       For further information see Comment tab!                        ***
 *********************************************************************************************)

// check if a start condition exists for the requested movement
bStartConditionOk := TRUE;
iStartConditionsNotOk := 0;
FOR i := 1 TO cMaxStartConditions DO
   IF sv_ODCSequence[StepPos.iColumn][StepPos.iRow] = sv_StartConditionInstanceData[i].DelayedMovement THEN
      // start condition found -> check if start condition is reached
      abInterpreter.aCheckStartConditionReached(iInstance := i);
      IF NOT abInterpreter.aCheckStartConditionReached.bReached THEN
         IF NOT bNoAlarms THEN
            // set alarm
            SET_ALARM(Name := erCompNotInCorrectPosition,
                      SubID1 := sv_StartConditionInstanceData[i].RelatedMovement.iCompId,
                      SubID2 := sv_StartConditionInstanceData[i].RelatedMovement.iIndexId);
         END_IF;
         bStartConditionOk := FALSE;
         iStartConditionsNotOk := iStartConditionsNotOk + 1;
      END_IF;
   ELSIF sv_ODCSequence[StepPos.iColumn][StepPos.iRow] = sv_StartConditionInstanceData[i].RelatedMovement THEN
      //also check if the requested movement is the "RelatedMovement" of a startcondition
      //for example: core in with startpos parallel to mold close
      //if mold close movement is requested, the core must be out until the start position for the core is reached

      //check if start condition is reached
      abInterpreter.aCheckStartConditionReached(iInstance := i);
      IF NOT abInterpreter.aCheckStartConditionReached.bReached THEN
         //check safety array
         abODCCheckDependencies.aCheck.StepPos.iColumn := mStartConditionPosArray[i].iColumn;
         abODCCheckDependencies.aCheck.StepPos.iRow := mStartConditionPosArray[i].iRow;

         abODCCheckDependencies.aCheck(DeviceIdSelf := sv_DeviceId, bNoAlarmsAndStepState := bNoAlarms);
         IF NOT abODCCheckDependencies.aCheck.bAllowed THEN
            fbDebugTrace2(nODCInterpreter, CONCAT('manual movement at pos ',
                                                   DINT_TO_STRING(StepPos.iRow),
                                                   '/',
                                                   DINT_TO_STRING(StepPos.iColumn),
                                                   ' not allowed because of related startcondition'));
            bStartConditionOk := FALSE;
            iStartConditionsNotOk := iStartConditionsNotOk + 1;
         END_IF;
      END_IF;
   END_IF;
END_FOR;

// check if a check condition exists for the requested movement
bCheckConditionsOk := TRUE;
bCheckConditionFound := FALSE;
iCheckConditionsNotOk := 0;
abInterpreter.aFindCheckCondition(Movement := sv_ODCSequence[StepPos.iColumn][StepPos.iRow],
                                    bFound => bCheckConditionFound);

IF bCheckConditionFound THEN
   abInterpreter.aCheckConditionsManual(Movement := sv_ODCSequence[StepPos.iColumn][StepPos.iRow], bNoAlarms := bNoAlarms);
   bCheckConditionsOk := abInterpreter.aCheckConditionsManual.bCheckConditionsOk;
   iCheckConditionsNotOk := abInterpreter.aCheckConditionsManual.iConditionsNotOk;
END_IF;

;#END_EDIT_BLOCK END_ALGORITHM

(*
Start a single movement (in response to evStartRequest)

Basically the same movement can occur more than one time in the machine sequence.
If the requested movement is found in the sequence and all conditions are ok, this movement is started.
If one or more conditions (safety conditions, start conditions, check conditions) are not ok, the
algorithm continues searching because possibly the movement is found again and the conditions for this step are ok.

If the movement is not allowed, the movement position with the lowest number of not fulfilled conditions is marked (step state is set)
and tha according alarms are set

*)

ALGORITHM aStartSingleMovement

VAR_INPUT
 DeviceId : tsDeviceId;
 MoveDir : tMoveIdent;
 MoveId : tMoveIdent;
 IntermediateCond : DINT;
 bNeedCheckSafety : BOOL;
END_VAR

VAR_OUTPUT
 bStarted : BOOL;
END_VAR

VAR_TEMP
 StepPos : tsODCStepPos;
 evCheckLocklistEventData : tevCheckLocklistData;
END_VAR

VAR
 fbStart : FBStart;
 abODCCheckDependenciesStart : ABODCCheckDependencies;
 bStartConditionOk : BOOL;
 bCheckConditionsOk : BOOL;
 bCheckConditionFound : BOOL;
 fbSetStepState : FBSetStepState;
 bIgnoreConditions : BOOL;
 bSearchMovement : BOOL;
 bMovementFound : BOOL;
 bMovementAllowed : BOOL;
 TmpStepPos : tsODCStepPos;
 iTmpAlarmCount : DINT;
 StepPosLowestAlarms : tsODCStepPos;
 iAlarmCount : DINT;
END_VAR
#BEGIN_EDIT_BLOCK
(**************************************** WARNING ********************************************
 *** The KEBA Kemro K2 System including software is not intended for safety control tasks! ***
 ***                       For further information see Comment tab!                        ***
 *********************************************************************************************)

bStarted := FALSE;
bMovementFound := FALSE;
bSearchMovement := TRUE;
iAlarmCount := 0;
TmpStepPos.iColumn := 1;
TmpStepPos.iRow := 1;

//core and ejector movements should be possible in "override" mode
//no matter if they are programmed in sequence or not
bIgnoreConditions := (((DeviceId.CompId = cCompCore) AND sv_bOverrideCoreSafety)) OR
                     (((DeviceId.CompId = cCompEjector) AND sv_bOverrideEjectorSafety));

WHILE bSearchMovement DO

   //search for the requested movement
   abInterpreter.aFindLabel.SearchStartPos := TmpStepPos;
   abInterpreter.aFindLabel(DeviceId := DeviceId, MoveId :=MoveId, MoveDir := MoveDir, IntermediateCond := IntermediateCond, bAllowNonMatchingId := FALSE);
   IF abInterpreter.aFindLabel.bFound THEN
      bMovementFound := TRUE;
      StepPos := abInterpreter.aFindLabel.StepPos;
   ELSE
      //movement not found in sequence
      bSearchMovement := FALSE;
      StepPos.iColumn := 0;
      StepPos.iRow := 0;
   END_IF;

   IF abInterpreter.aFindLabel.bFound OR NOT bNeedCheckSafety OR bIgnoreConditions THEN
      //check conditions for this movement
      abODCCheckDependenciesStart.aCheck(StepPos := StepPos, DeviceIdSelf := DeviceId, bNoAlarmsAndStepState := TRUE);

      // check existing start conditions and check conditions for the requested movement
      // attention: check is only necessary if sequence is programmed by editor
      bStartConditionOk := TRUE;
      bCheckConditionsOk := TRUE;
      bCheckConditionFound := FALSE;

      IF NOT bIgnoreConditions THEN
         IF NOT sv_bUseProgramSwitches AND bNeedCheckSafety AND abInterpreter.aFindLabel.bFound THEN
            aStartAndCheckConditions(StepPos := StepPos,
                                     bNoAlarms := TRUE,
                                     bStartConditionOk => bStartConditionOk,
                                     bCheckConditionsOk => bCheckConditionsOk,
                                     bCheckConditionFound => bCheckConditionFound);
         END_IF;
      END_IF;

      iTmpAlarmCount := 0;
      IF NOT abODCCheckDependenciesStart.aCheck.bAllowed THEN
         //safety conditions not ok => save number of not fulfilled conditions
         iTmpAlarmCount := abODCCheckDependenciesStart.aCheck.iNotOkCount;
      END_IF;

      IF NOT bStartConditionOk THEN
         //start conditions not ok => increment nummber of not fulfilled conditions
         iTmpAlarmCount := iTmpAlarmCount + aStartAndCheckConditions.iStartConditionsNotOk;
      END_IF;

      IF NOT bCheckConditionsOk THEN
         //check conditions not ok => increment nummber of not fulfilled conditions
         iTmpAlarmCount := iTmpAlarmCount + aStartAndCheckConditions.iCheckConditionsNotOk;
      END_IF;

      //everything OK -> start movement and exit loop
      IF abODCCheckDependenciesStart.aCheck.bAllowed AND bStartConditionOk AND bCheckConditionsOk THEN
         //movement with correct condition found => start this movement
         abInterpreter.aAddStartedManualMovement(DeviceId := DeviceId, MoveId := MoveId, MoveDir := MoveDir,
                                                 StepPos := StepPos, iInstance := IntermediateCond);
         IF abInterpreter.aAddStartedManualMovement.bOK THEN
            fbStart(DeviceId := DeviceId, MoveDir := MoveDir, MoveId := MoveId, IntermediateCond := IntermediateCond);
            bStarted := TRUE;

            //set step state to active
            IF (StepPos.iColumn <> 0) AND (StepPos.iRow <> 0) THEN
               fbSetStepState(StepPos := StepPos,
                              StepState := nStateActive);
            END_IF;
         END_IF;

         IF bCheckConditionFound THEN
            START_PROCESS_ALGORITHM(paCheckConditionsManual);
         END_IF;

         IF NOT abInterpreter.aFindLabel.bFound THEN
            fbDebugTrace2(nODCInterpreter, 'Manual Movement started anyway because it is not safety relevant');
         END_IF;

         bSearchMovement := FALSE;
         bMovementAllowed := TRUE;
         RETURN; // ******  exit algorithm *******
      ELSE
         //check number of not fulfilled conditions
         IF (iAlarmCount = 0) OR (iTmpAlarmCount < iAlarmCount) THEN
            //save this step
            StepPosLowestAlarms := StepPos;
            iAlarmCount := iTmpAlarmCount;
            iTmpAlarmCount := 0;
         END_IF;

         //save this position (needed as startposition of next search)
         //attention: iColumn must be increased otherwise always the same step will be found
         TmpStepPos.iColumn := StepPos.iColumn + 1;
         TmpStepPos.iRow := StepPos.iRow;
         bMovementAllowed := FALSE;
      END_IF;
   END_IF;  //end_if aFindLabel.bFound

END_WHILE;

IF NOT bMovementFound THEN
   fbDebugTrace2(nODCInterpreter, 'Manual Movement not started because movement is safety relevant but not in ODC');
ELSIF NOT bMovementAllowed THEN
   //use step which causes the lowest number of alarms
   //call dependency check again to set the according alarms
   abODCCheckDependenciesStart.aCheck(StepPos := StepPosLowestAlarms, DeviceIdSelf := DeviceId, bNoAlarmsAndStepState := FALSE);

   //set alarms related to start and check conditions
   aStartAndCheckConditions(StepPos := StepPosLowestAlarms,
                            bNoAlarms := FALSE,
                            bStartConditionOk => bStartConditionOk,
                            bCheckConditionsOk => bCheckConditionsOk,
                            bCheckConditionFound => bCheckConditionFound);

   //set step state to error
   fbSetStepState(StepPos := StepPosLowestAlarms, StepState := nStateError);

   //evCheckLocklist makes sure other alarms(caused by FBLockUnlock for this movement are also set *)
   fbDebugTrace2(nODCInterpreter, CONCAT('Manual Movement ', DINT_TO_STRING(MoveId),
                                          '/', DINT_TO_STRING(MoveDir),
                                          ' not started because safety conditions do not allow it -> sending evCheckLocklist to view all other alarms'));
   evCheckLocklistEventData.DeviceId := DeviceId;
   evCheckLocklistEventData.MoveId   := MoveId;
   evCheckLocklistEventData.MoveDir  := MoveDir;
   SET_EVENT(evCheckLocklist, evCheckLocklistEventData);

   IF NOT bStartConditionOk THEN
      fbDebugTrace2(nODCInterpreter, 'Manual Movement not started because start condition not ok');
   END_IF;

   IF NOT bCheckConditionsOk THEN
      fbDebugTrace2(nODCInterpreter, 'Manual Movement not started because check condition not ok');
   END_IF;
END_IF;

;#END_EDIT_BLOCK END_ALGORITHM

(*
Start a combined movement (in response to evStartRequest)
*)

ALGORITHM aStartCombinedMovement

VAR_INPUT
 DeviceId : tsDeviceId;
 MoveDir : tMoveIdent;
 MoveId : tMoveIdent;
END_VAR

VAR_OUTPUT
 bNotFound : BOOL;
END_VAR

VAR_TEMP
 StartPos : tsODCStepPos;
END_VAR
#BEGIN_EDIT_BLOCK
(**************************************** WARNING ********************************************
 *** The KEBA Kemro K2 System including software is not intended for safety control tasks! ***
 ***                       For further information see Comment tab!                        ***
 *********************************************************************************************)

bNotFound := FALSE;

(* find start label *)
abInterpreter.aFindLabel.SearchStartPos.iColumn := 1;
abInterpreter.aFindLabel.SearchStartPos.iRow := 1;
abInterpreter.aFindLabel(DeviceId := DeviceId,
                         MoveId := cMoveBeginSequence,
                         MoveDir := MoveDir,
                         IntermediateCond := 0,
                         bAllowNonMatchingId := FALSE);
IF NOT abInterpreter.aFindLabel.bFound THEN
   fbDebugTrace2(nODCInterpreter, 'combined movement -> start label not found -> will try to start single movement');
   bNotFound := TRUE;
   RETURN;
END_IF;

StartPos := abInterpreter.aFindLabel.StepPos;

(* find end of label *)
abInterpreter.aFindLabel(DeviceId := DeviceId,
                         MoveId := cMoveEndSequence,
                         MoveDir := MoveDir,
                         IntermediateCond := 0,
                         bAllowNonMatchingId := FALSE);
IF NOT abInterpreter.aFindLabel.bFound THEN
   fbDebugTrace2(nODCInterpreter, 'combined movement -> end label not found -> will try to start single movement');
   bNotFound := TRUE;
   RETURN;
END_IF;

// save active sequence (for highlighting in machine sequencer)
sv_ActiveSequence.DeviceId := DeviceId;
sv_ActiveSequence.MoveDir := MoveDir;
sv_ActiveSequence.iCount :=  sv_ActiveSequence.iCount + 1;
sv_ActiveSequence.bActive := TRUE;

(* remember for later so we can stop combined movements *)
mStartedCombinedMovement.DeviceId := DeviceId;
mStartedCombinedMovement.MoveId   := MoveId;
mStartedCombinedMovement.MoveDir  := MoveDir;

abInterpreter.aInitInterpreter(iColumn := StartPos.iColumn,
                               iRow := StartPos.iRow,
                               iEndRow := abInterpreter.aFindLabel.StepPos.iRow,
                               bSkipAlreadyPosReached := TRUE,
                               bExcludeActiveColumns := FALSE);

(* paRunManualCombinedMovement stops itself when interpreter is not active anymore *)
START_PROCESS_ALGORITHM(paRunManualCombinedMovement);

;#END_EDIT_BLOCK END_ALGORITHM

(*
Handle evStartRequest(manual buttons)
start requests will be ignored in the following situations:
- sequence array not initialized completely
  (startup or creation of new sequence in progress, creation of sequence failed)
- machine running in half or fullauto cycle
- teachmode in machine sequencer is active
*)

EVENT_ALGORITHM evaStartRequest ON EV_Task_3(23) WITH evStartRequest

VAR_INPUT
 evStartRequestData : tevStartRequestData;
END_VAR

VAR_TEMP
 i : DINT;
END_VAR

VAR
 StartRequestData : tevStartRequestData;
 bCheckSafety : BOOL;
 iSafety : DINT;
 bCombined : BOOL;
END_VAR
#BEGIN_EDIT_BLOCK
(**************************************** WARNING ********************************************
 *** The KEBA Kemro K2 System including software is not intended for safety control tasks! ***
 ***                       For further information see Comment tab!                        ***
 *********************************************************************************************)

IF mbRecalcActive THEN
   //Ignore start requests if a cycle recalc is active.
   //This flag is set by aDoPendingRecalc() before the low priority paInitSequence actually starts executing code
   //This is necessary to avoid problems where a recalc and a movement start happen at the same cycle
   fbDebugTrace2(nDeviceState, 'evStartRequest ignored because sequence is being recalculated');
   RETURN;
END_IF;

IF sv_iInitOK <> 20 THEN
   //ignore start requests if array is not initialized completely
   //this can happen during startup and during creation of a new sequence
   //or if creation of a sequence failed
   fbDebugTrace2(nDeviceState, 'evStartRequest ignored because sequence not initialized');
   RETURN;
END_IF;

IF sv_OperationMode >= nHalfAutomatic THEN
   IF sv_bSequenceInterruption THEN
      //sequence is actually interrupted -> find out if it is allowed to start this movement
      fbGetMoveNumber(DeviceId := evStartRequestData.DeviceId,
                     MoveDir := evStartRequestData.MoveDir,
                     MoveId := evStartRequestData.MoveId);

      IF fbGetMoveNumber.bFound THEN
         IF sv_MovementsAvailable[fbGetMoveNumber.iMoveNumber].pMovementData^.bAllowedDuringInterrupt THEN
            //try to start this movement
            aStartSingleMovement(DeviceId := evStartRequestData.DeviceId,
                                 MoveDir := evStartRequestData.MoveDir,
                                 MoveId := evStartRequestData.MoveId,
                                 IntermediateCond := evStartRequestData.IntermediateCond,
                                 bNeedCheckSafety := FALSE);
         END_IF;
      END_IF;
   ELSE
      //ignore start requests if operation mode is half or full automatic
      fbDebugTrace2(nDeviceState, 'evStartRequest ignored because in half or full auto mode');
   END_IF;

   RETURN; // return here
END_IF;

IF sv_iActiveEditors > 0 THEN
   //teach mode active -> ignore start requests
   SET_ALARM(Name := erTeachModeActive);
   RETURN;
END_IF;

StartRequestData := evStartRequestData;

// work with StartRequest
fbGetMoveNumber(DeviceId := StartRequestData.DeviceId,
                MoveDir := StartRequestData.MoveDir,
                MoveId := StartRequestData.MoveId);

IF fbGetMoveNumber.bFound THEN
   iSafety := sv_MovementsAvailable[fbGetMoveNumber.iMoveNumber].pMovementData^.iSafetyIdentifier;
   (* FIXME: always set the intermediate condition to 0 when movement does not have intermediate conditions
      needed for searching the movement
   *)
   IF NOT sv_MovementsAvailable[fbGetMoveNumber.iMoveNumber].pMovementData^.bInstanceable THEN
      StartRequestData.IntermediateCond := 0;
   END_IF;
ELSE
   fbDebugTrace2(nODCInterpreter, 'could not find movement -> assuming movement is safety relevant');
   iSafety := 1;
END_IF;

IF iSafety = 1 THEN
   bCheckSafety := TRUE;
   fbDebugTrace2(nODCInterpreter, 'movement is safety relevant (sequence safety and mold safety (safety editor)');
ELSIF iSafety = 3 THEN
   bCheckSafety := TRUE;
   fbDebugTrace2(nODCInterpreter, 'movement is safety relevant (sequence safety only - no mold safety (safety editor)');
ELSIF iSafety = 2 THEN
   // only check pos reached of other movements, movement itself is not safety relevant
   bCheckSafety := TRUE;
   fbDebugTrace2(nODCInterpreter, 'movement is partially safety relevant');
ELSIF iSafety = 0 THEN
   bCheckSafety := FALSE;
   fbDebugTrace2(nODCInterpreter, 'movement is NOT safety relevant');
ELSE
   bCheckSafety := TRUE;
   fbDebugTrace(CONCAT('strange safety relevance value ', DINT_TO_STRING(iSafety)));
END_IF;

abInterpreter.aStatus();
IF abInterpreter.aStatus.bActive THEN
   fbDebugTrace2(nODCInterpreter, 'manual movement not started because there is already a combined movement active');

   SET_ALARM(Name := erMovementDuringActiveSequence,
             SubID1 := StartRequestData.DeviceId.CompId,
             SubID2 := StartRequestData.MoveId,
             SubID3 := mStartedCombinedMovement.DeviceId.CompId,
             SubID4 := mStartedCombinedMovement.MoveId,
             Param1 := DINT_TO_STRING(StartRequestData.DeviceId.IndexId));
   RETURN;
END_IF;

(* Rules:
 * When a combined movement is active no other movement may be started
 * When any movement is active no combined movement may be started
 * Autopurge counts as 1 or more movementy so the above rule covers this already
   -> single movements are allowed during autopurge
 * When operation mode is setup, combined movement are never started(only single movemets *)

IF sv_bCombinedMovementsInManual AND (StartRequestData.MoveId = cMoveBeginSequence) THEN
   IF sv_OperationMode = nSetup THEN
      fbDebugTrace2(nODCInterpreter, 'starting a combined movement in setup mode is not allowed');
      RETURN;
   END_IF;
   bCombined := TRUE;
ELSIF sv_bCombinedMovementsInManual AND (sv_OperationMode = nManual) AND
   (* combined movements are not allowed in setup mode *)
   (StartRequestData.DeviceId.CompId = cCompMold AND
   ((StartRequestData.MoveDir = cMoveFwd OR
    StartRequestData.MoveDir = cMoveBwd))
   OR
   (StartRequestData.DeviceId.CompId = cCompInjection AND
   (StartRequestData.MoveId = cMoveInject OR
    StartRequestData.MoveId = cMoveCombinedPlast))) THEN
   //this check is for MoveId as plasticize, decompress and intrusion have MoveDir = cMoveBwd
   bCombined := TRUE;
ELSE
   bCombined := FALSE;

   //check if  requested device is activated
   FOR i := 1 TO sv_ODCDeviceMovements.iCount DO
      IF sv_ODCDeviceMovements.Devices[i].DeviceId = StartRequestData.DeviceId THEN
         IF NOT sv_ODCDeviceMovements.Devices[i].pbDeviceActivated^ THEN
            fbDebugTrace2(nODCInterpreter, 'start request ignored because device is not activated');
            RETURN;
         END_IF;
         EXIT;
      END_IF;
   END_FOR;
END_IF;

IF sv_StartedMovements.iStartedMovements <> 0 AND bCombined THEN
   fbDebugTrace2(nODCInterpreter, 'combined manual movement not started because there is already a movement active');

   SET_ALARM(Name := erSequenceDuringActiveMovement,
             SubID1 := StartRequestData.DeviceId.CompId,
             SubID2 := StartRequestData.DeviceId.IndexId,
             SubID3 := StartRequestData.MoveId);
   RETURN;
END_IF;

(* back up sequence when a movement is started
   and the sequence has changed *)
START_PROCESS_ALGORITHM(paBackupSequence);

IF bCombined THEN
   fbDebugTrace2(nODCInterpreter, 'evStartRequest -> starting a combined movement');
   aClearStepState(FALSE);
   aStartCombinedMovement(DeviceId := StartRequestData.DeviceId,
                          MoveDir := StartRequestData.MoveDir,
                          MoveId := StartRequestData.MoveId);
END_IF;

IF NOT bCombined OR aStartCombinedMovement.bNotFound THEN
   (* if combined movement markers were not found start single movement *)
   IF (StartRequestData.MoveId = cMoveBeginSequence) THEN
      //do not try to start a single movement if a start request for
      //cMoveBeginSequence was received and this sequence was not found
      fbDebugTrace2(nODCInterpreter, 'requested combined movement not found');
   ELSE
      fbDebugTrace2(nODCInterpreter, 'evStartRequest -> starting a single movement');
      aStartSingleMovement(DeviceId := StartRequestData.DeviceId,
                           MoveDir := StartRequestData.MoveDir,
                           MoveId := StartRequestData.MoveId,
                           IntermediateCond := StartRequestData.IntermediateCond,
                           bNeedCheckSafety := bCheckSafety);
   END_IF;
END_IF;

;#END_EDIT_BLOCK END_ALGORITHM

(*
Handle evStopRequest(manual buttons)
Stop single and combined movements
*)

EVENT_ALGORITHM evaStopRequest ON EV_Task_3 WITH evStopRequest

VAR_INPUT
 evStopRequestData : tevStopRequestData;
END_VAR

VAR
 fbStop : FBStop;
END_VAR
#BEGIN_EDIT_BLOCK
(**************************************** WARNING ********************************************
 *** The KEBA Kemro K2 System including software is not intended for safety control tasks! ***
 ***                       For further information see Comment tab!                        ***
 *********************************************************************************************)

IF NOT sv_bInitDone THEN
   //ignore stop requests before sv_bInitDone
   fbDebugTrace2(nDeviceState, 'evStopRequest ignored because sv_bInitDone is not TRUE');
   RETURN;
END_IF;

IF (sv_OperationMode >= nHalfAutomatic) AND NOT sv_bSequenceInterruption THEN
   //ignore stop requests if operation mode is half or full automatic
   //stop requests for movements which were started during sequence interruption
   //must be handled
   fbDebugTrace2(nDeviceState, 'evStopRequest ignored because in half or full auto mode');
   RETURN;
END_IF;

abInterpreter.aStatus();
IF abInterpreter.aStatus.bActive THEN
   IF mStartedCombinedMovement.DeviceId = evStopRequestData.DeviceId AND
      mStartedCombinedMovement.MoveId = evStopRequestData.MoveId AND
      mStartedCombinedMovement.MoveDir = evStopRequestData.MoveDir THEN
      // we get a stop request for the combined movement
      // so stop it
      fbDebugTrace2(nDeviceState, 'evStopRequest while interpreter is active -> aStopInterpreterNormal()');
      abInterpreter.aStopInterpreterNormal();
      sv_ActiveSequence.bActive := FALSE;
   ELSE
      // we get a stop request for a single movement
      // but a combined movement is active
      // but no single movements are allowed during a combined movement
      // -> ignore the event
      fbDebugTrace2(nDeviceState, 'evStopRequest ignored because combined movement is active and device/movement does not match');
   END_IF;
ELSE
   fbDebugTrace2(nDeviceState, 'evStopRequest while interpreter is inactiveactive -> fbStop()');
   // it is also possible that the interpreter already finished the combined movement
   // we still send a evStop, but that does not cause ony problems
   fbStop(DeviceId := evStopRequestData.DeviceId);
   sv_ActiveSequence.bActive := FALSE;
END_IF;

// no movenumber available, clear all
g_SafetyData.MovementToActivate := 0;

;#END_EDIT_BLOCK END_ALGORITHM

ALGORITHM aDecreaseLineNumber

VAR_INPUT
 DeviceId : tsDeviceId;
 MoveId : tMoveIdent;
 MoveDir : tMoveIdent;
END_VAR

VAR_TEMP
 iTmpColumn : DINT;
 i : DINT;
END_VAR

VAR
 fbCheckPosReached : FBCheckPosReached;
 dummy : DINT;
END_VAR
#BEGIN_EDIT_BLOCK
(**************************************** WARNING ********************************************
 *** The KEBA Kemro K2 System including software is not intended for safety control tasks! ***
 ***                       For further information see Comment tab!                        ***
 *********************************************************************************************)

FOR i := 1 TO sv_iUsedColumns DO
   IF (mActiveStepBwdMovements[i].DeviceId = DeviceId) AND
      (mActiveStepBwdMovements[i].MoveId = MoveId) AND
      (mActiveStepBwdMovements[i].MoveDir = MoveDir) THEN

      //check posReached flag
      fbCheckPosReached(DeviceId := DeviceId,
                        MoveDir := MoveDir,
                        MoveId := MoveId);

      IF CHECK_REF(fbCheckPosReached.pbPosReached^) AND NOT fbCheckPosReached.pbPosReached^ THEN
         ;//endposition not reached -> do not decrease line number
      ELSE
         //endposition reached or no posReached flag available -> decrease row
         iTmpColumn := i;
         REPEAT
            IF sv_TraceLevel.bODCInterpreter THEN
               dummy := Print('call abInterpreter.aDecreaseRow with iColumn = %d', iTmpColumn);
            END_IF;
            abInterpreter.aDecreaseRow(bStartInActualLine := FALSE,
                                       iColumn := iTmpColumn,
                                       iEndRow := 1);
            iTmpColumn := abInterpreter.aDecreaseRow.iNewActivatedColumn;

         UNTIL (abInterpreter.aDecreaseRow.iNewActivatedColumn = 0)
         END_REPEAT;
      END_IF;

      //init this element
      mActiveStepBwdMovements[i].DeviceId.CompId := cCompNone;
      mActiveStepBwdMovements[i].DeviceId.IndexId := 1;
      mActiveStepBwdMovements[i].MoveId := cMinMoveIdent;
      mActiveStepBwdMovements[i].MoveDir := cMoveNone;

      EXIT;
   END_IF;
END_FOR;

;#END_EDIT_BLOCK END_ALGORITHM

(*
Manage list and count of currently started movments
in sv_StartedMovements when receiving evStartedStopped events
*)

EVENT_ALGORITHM evaStartedStopped ON EV_Task_3 WITH evStartedStopped

VAR_INPUT
 evStartedStoppedData : tevStartedStoppedData;
END_VAR

VAR_TEMP
 tmpMovement : tsStartedMoveInfoODCExtended;
 i : DINT;
 stepPos : tsODCStepPos;
 idx : DINT;
END_VAR

VAR
 bFound : BOOL;
 fbSetStepState : FBSetStepState;
 bCorrectInstance : BOOL;
END_VAR
#BEGIN_EDIT_BLOCK
(**************************************** WARNING ********************************************
 *** The KEBA Kemro K2 System including software is not intended for safety control tasks! ***
 ***                       For further information see Comment tab!                        ***
 *********************************************************************************************)

IF evStartedStoppedData.State = nStopped OR  evStartedStoppedData.State = nStartNotAllowed THEN
   bFound := FALSE;
   // movement was stopped or never started
   // remove movement from list with started movements

   Status := MovementsSema.Wait(WaitTime := cTimeOutSempahore);
   IF Status <> KRTOS_Status_OK THEN
      dummy2 := ASSERT(FALSE, erAssert);
      RETURN;
   END_IF;

   FOR i := 1 TO sv_StartedManualMovements.iStartedMovements DO

      bCorrectInstance := (evStartedStoppedData.iInstance = 0) OR (evStartedStoppedData.iInstance = sv_StartedManualMovements.MoveData[i].iInstance);
      IF sv_StartedManualMovements.MoveData[i].DeviceId = evStartedStoppedData.DeviceId AND
         sv_StartedManualMovements.MoveData[i].MoveDir = evStartedStoppedData.MoveDir AND
         sv_StartedManualMovements.MoveData[i].MoveId = evStartedStoppedData.MoveId AND bCorrectInstance THEN

         stepPos := sv_StartedManualMovements.MoveData[i].StepPos;
         IF (g_SafetyData.bAvailable) THEN
            IF (NOT((stepPos.iColumn = 0) OR (stepPos.iRow = 0)))THEN
               idx := sv_MovementsAvailable[sv_ODCSequenceInt[stepPos.iColumn][stepPos.iRow].iMoveNumber].iODCSafetyMovementsEntry;
               IF (idx > 0) THEN
                  g_SafetyData.MovementToActivate := g_SafetyData.MovementToActivate AND (NOT SHL(1, idx-1));
               END_IF;
            END_IF;
         END_IF;

         IF (NOT((stepPos.iColumn = 0) OR (stepPos.iRow = 0)))THEN
            //only correct step sate if actual state is not error
            IF sv_ODCSequenceInt[stepPos.iColumn, stepPos.iRow].StepState <> nStateError THEN
               fbSetStepState(StepPos := sv_StartedManualMovements.MoveData[i].StepPos,
                           StepState := nStateReady);
            END_IF;

         END_IF;

         IF sv_TraceLevel.bODCInterpreter THEN
            dummy := Print('removing started manual movement %d.%d %d/%d', evStartedStoppedData.DeviceId.CompId, evStartedStoppedData.DeviceId.IndexId, evStartedStoppedData.MoveId, evStartedStoppedData.MoveDir);
         END_IF;

         //copy last entry in the list to this empty field
         sv_StartedManualMovements.MoveData[i] := sv_StartedManualMovements.MoveData[sv_StartedManualMovements.iStartedMovements];

         //zero last entry
         tmpMovement.DeviceId.CompId := cCompNone;
         tmpMovement.DeviceId.IndexId := 1;
         tmpMovement.MoveDir := cMoveNone;
         tmpMovement.MoveId := cMinMoveIdent;
         tmpMovement.StepPos.iColumn := 0;
         tmpMovement.StepPos.iRow := 0;
         tmpMovement.iInstance := 0;
         sv_StartedManualMovements.MoveData[sv_StartedManualMovements.iStartedMovements] := tmpMovement;

         sv_StartedManualMovements.iStartedMovements := sv_StartedManualMovements.iStartedMovements - 1;
         //fbDebugTrace2(nODCInterpreter, 'end removing started manual movement');
         bFound := TRUE;
         EXIT;
      END_IF;
   END_FOR;

   Status := MovementsSema.Put();
   IF Status <> KRTOS_Status_OK THEN
      dummy2 := ASSERT(FALSE, erAssert);
   END_IF;

   IF sv_bSequenceInterruption THEN
      //started / stopped event during sequence is interrupted
      //-> check if line number should be decreased
      aDecreaseLineNumber(DeviceId := evStartedStoppedData.DeviceId,
                          MoveId := evStartedStoppedData.MoveId,
                          MoveDir := evStartedStoppedData.MoveDir);
   END_IF;

   IF NOT bFound THEN
      IF sv_TraceLevel.bODCInterpreter THEN
         dummy := Print('tried to remove stopped movement, but not in list anymore???');
      END_IF;
   END_IF;
END_IF;

;#END_EDIT_BLOCK END_ALGORITHM

(*
Start / stop paCyclicConditionCheck depending on
if there are started movements.
*)

POSTUPDATE_ALGORITHM pStartedMovements ON PU_Task_3 WITH sv_StartedManualMovements.iStartedMovements

#BEGIN_EDIT_BLOCK
(**************************************** WARNING ********************************************
 *** The KEBA Kemro K2 System including software is not intended for safety control tasks! ***
 ***                       For further information see Comment tab!                        ***
 *********************************************************************************************)

IF sv_StartedManualMovements.iStartedMovements = 0 THEN
   STOP_PROCESS_ALGORITHM(paCyclicConditionCheck);
   STOP_PROCESS_ALGORITHM(paCheckConditionsManual);

   abInterpreter.aStatus();
   IF sv_OperationMode <= nManual AND NOT abInterpreter.aStatus.bActive THEN
      (* the last single manual movement was stopped -> recalculate if needed *)
      aDoPendingRecalc();
      IF aDoPendingRecalc.bStartedRecalc THEN
         fbDebugTrace2(nDeviceState, 'recalc because iStartedMovements = 0');
      END_IF;
   END_IF;
ELSE
   START_PROCESS_ALGORITHM(paCyclicConditionCheck);

END_IF;

;#END_EDIT_BLOCK END_ALGORITHM

(*
Cyclically check movement conditions of all started movements
(auto mode, combined manual movements, single manual movements)
*)

PROCESS_ALGORITHM paCyclicConditionCheck ON TaskAnalog

VAR_TEMP
 i : DINT;
END_VAR

VAR
 abODCCheckDependenciesCyclic : ABODCCheckDependencies (* must be a separate block since it is accessed from different tasks at the same time *);
 TmpStepPos : tsODCStepPos;
END_VAR
#BEGIN_EDIT_BLOCK
(**************************************** WARNING ********************************************
 *** The KEBA Kemro K2 System including software is not intended for safety control tasks! ***
 ***                       For further information see Comment tab!                        ***
 *********************************************************************************************)

abInterpreter.aStatus();

Status := MovementsSema.Wait(WaitTime := cTimeOutSempahore);
IF Status <> KRTOS_Status_OK THEN
   dummy2 := ASSERT(FALSE, erAssert);
   RETURN;
END_IF;

FOR i := 1 TO sv_StartedManualMovements.iStartedMovements DO
   // check safety for manual movements
   // abODCCheckSafetyConditions must be a separete instance
   // because this PROCESS_ALGORITHM runs in a fast task that can
   // interrupt other tasks
   TmpStepPos := sv_StartedManualMovements.MoveData[i].StepPos;
   IF(abInterpreter.aStatus.bActive AND (TmpStepPos.iColumn = 0 OR TmpStepPos.iRow = 0)) THEN
      fbDebugTrace('interpreter is active but a movement with step pos 0 is running'); //this might be legitime, but is most times not normal
      abInterpreter.aStopInterpreterFatal();
   END_IF;

   abODCCheckDependenciesCyclic.aCheck(StepPos := TmpStepPos, DeviceIdSelf := sv_StartedManualMovements.MoveData[i].DeviceId);
   IF NOT abODCCheckDependenciesCyclic.aCheck.bAllowed THEN
      fbDebugTrace2(nODCInterpreter, CONCAT('cyclic condition check reported movement at ',
                                            DINT_TO_STRING(sv_StartedManualMovements.MoveData[i].StepPos.iColumn),
                                            '/',
                                            DINT_TO_STRING(sv_StartedManualMovements.MoveData[i].StepPos.iRow),
                                            ' as not allowed'));
      abInterpreter.aStopInterpreterError();
   END_IF;

END_FOR;

//FIXME: is it a good idea to hold the lock so long???
Status := MovementsSema.Put();
IF Status <> KRTOS_Status_OK THEN
   dummy2 := ASSERT(FALSE, erAssert);
END_IF;

;#END_EDIT_BLOCK END_ALGORITHM

(*
Run the autocycle by calling the interpreter.
*)

ALGORITHM aRunAutoCycle

VAR_INPUT
 bStopCycle : BOOL (* stop cycle immediately *);
 bStopAfterCycle : BOOL (* finish the actual cycle and stop *);
END_VAR

VAR_OUTPUT
 bReady : BOOL;
END_VAR

VAR
 bCanStart : BOOL (* got the cycle start signal-> cycle can start if sequence recalc is finished *);
 abWaitCycleStart : ABWaitCycleStart;
 fbStart : FBStart;
 bDelayExceeded : BOOL;
 bEjectorBwdStarted : BOOL;
 DeviceIdEjector : tsDeviceId := (CompId:=cCompEjector,IndexId:=1);
 bInitDone : BOOL;
 pbEjectorBwd : REFTO BOOL;
 pbEjectorBwdActivated : REFTO BOOL;
 pbEjectorReady : REFTO BOOL;
 iMoveNrEjectorBwd : DINT;
 bColumnActive : BOOL;
 bDoRecalc : BOOL;
 bMovesBeforeAutoLoop : BOOL;
END_VAR

(* IecGraph-Code *)

(* init step *)
INITIAL_STEP S_CheckStartCond:
AAutoCycleReady (P);
END_STEP

ACTION AAutoCycleReady: #BEGIN_EDIT_BLOCK
bReady := TRUE;
IF (sv_OperationMode <> nFullAutomatic) THEN
   sv_bAutoCycleRunning := FALSE;
END_IF;
g_SafetyData.MovementToActivate := 0;
abInterpreter.aResetStepMode();

;#END_EDIT_BLOCK END_ACTION (*AAutoCycleReady*)

(* steps *)
STEP S_CheckStartCycle:
AAutoInit (P);
AWaitCycleStart (N);
aRecalc (N);
ADelayCycle (N);
END_STEP

ACTION AAutoInit: #BEGIN_EDIT_BLOCK
bReady := FALSE;
IF (sv_OperationMode <> nFullAutomatic) THEN
   sv_bAutoCycleRunning := FALSE;
END_IF;
bCanStart := FALSE;
abWaitCycleStart.aCycleStartRequest();

;#END_EDIT_BLOCK END_ACTION (*AAutoInit*)
ACTION AWaitCycleStart: #BEGIN_EDIT_BLOCK
abWaitCycleStart.aWaitCycleStart();
IF abWaitCycleStart.aWaitCycleStart.bCanStart THEN
   (* save flag because it is only TRUE for 1 cycle *)
   bCanStart := TRUE;
END_IF;

;#END_EDIT_BLOCK END_ACTION (*AWaitCycleStart*)
ACTION aRecalc: #BEGIN_EDIT_BLOCK
// allow to recalculate the cycle while waiting for the start signal
// but delay real start of the sequence until recalculation is finished
aDoPendingRecalc();
IF aDoPendingRecalc.bStartedRecalc THEN
   fbDebugTrace2(nDeviceState, 'recalc because autocycle start wait');
END_IF;

;#END_EDIT_BLOCK END_ACTION (*aRecalc*)
STEP Step42:
END_STEP

STEP Step43:
END_STEP

STEP Step44:
AMovementsBeforeCycleLoop (P);
END_STEP

ACTION AMovementsBeforeCycleLoop: #BEGIN_EDIT_BLOCK
IF (g_iAutoCycleLoopStartLine > 2) THEN
   bMovesBeforeAutoLoop := TRUE;
ELSE
   bMovesBeforeAutoLoop := FALSE;
END_IF;

;#END_EDIT_BLOCK END_ACTION (*AMovementsBeforeCycleLoop*)
STEP Step20:
END_STEP

STEP S_EjectorAutoBwd:
AInitEjectorBwd (P);
AEjectorAutoBwd (P);
END_STEP

STEP S_CheckEjectorBwd:
ACheckEjectorBwd (P);
END_STEP

STEP S_BeforeCycleLoop:
AStepsBeforeCycle (P);
ARunStepsBeforeCycle (N);
END_STEP

ACTION AStepsBeforeCycle: #BEGIN_EDIT_BLOCK
aClearStepState(FALSE);
abInterpreter.aInitInterpreter(iColumn := 1,
                               iRow := 1,
                               iEndRow := g_iAutoCycleLoopStartLine,
                               bSkipAlreadyPosReached := FALSE,
                               bExcludeActiveColumns := FALSE);

abInterpreter.aIncreaseRow(iColumn := 1,
                           iEndRow := g_iAutoCycleLoopStartLine);

;#END_EDIT_BLOCK END_ACTION (*AStepsBeforeCycle*)
ACTION ARunStepsBeforeCycle: #BEGIN_EDIT_BLOCK
abInterpreter.aInterpret();
abInterpreter.aStatus();

;#END_EDIT_BLOCK END_ACTION (*ARunStepsBeforeCycle*)
STEP S_ODC1:
AStartCycle (P);
AInitInterpreter (P);
END_STEP

STEP S_Run:
ARunInterpreter (N);
END_STEP

ACTION ARunInterpreter: #BEGIN_EDIT_BLOCK
abInterpreter.aInterpret();
abInterpreter.aStatus();

;#END_EDIT_BLOCK END_ACTION (*ARunInterpreter*)
STEP SErrorWait:
AAutoManual (N);
END_STEP

ACTION AAutoManual: #BEGIN_EDIT_BLOCK
fbAutoManual();

;#END_EDIT_BLOCK END_ACTION (*AAutoManual*)
STEP S_FinishCycle:
AIncreaseShotCounter (P);
AResetFlags (P);
END_STEP

ACTION AIncreaseShotCounter: #BEGIN_EDIT_BLOCK
g_SafetyData.MovementToActivate := 0;

fbStart.DeviceId.CompId := cCompOperationMode;
fbStart.DeviceId.IndexId := 1;
fbStart.MoveDir := cMoveNone;
fbStart.MoveId := cMoveIncreaseShotCounter;
fbStart();

;#END_EDIT_BLOCK END_ACTION (*AIncreaseShotCounter*)
ACTION AResetFlags: #BEGIN_EDIT_BLOCK
sv_bFirstCycle := FALSE;
mbCycleTimeMachineRunning := FALSE;

;#END_EDIT_BLOCK END_ACTION (*AResetFlags*)
STEP S_CheckStopCycle:
ACheckRecalcPending (P);
END_STEP

ACTION ACheckRecalcPending: #BEGIN_EDIT_BLOCK
bDoRecalc := (mPendingRecalc <> nODCRecalcNone)

;#END_EDIT_BLOCK END_ACTION (*ACheckRecalcPending*)
STEP Step27:
ACheckColumnActive (P);
END_STEP

ACTION ACheckColumnActive: #BEGIN_EDIT_BLOCK
aIsAnyColumnActive(bActive => bColumnActive);

;#END_EDIT_BLOCK END_ACTION (*ACheckColumnActive*)
STEP S_FinishParallelOpen:
AFinishParallelOpen (N);
ACheckColumns (N);
END_STEP

ACTION AFinishParallelOpen: #BEGIN_EDIT_BLOCK
//call interpreter until all columns
//are finished
abInterpreter.aInterpret();

;#END_EDIT_BLOCK END_ACTION (*AFinishParallelOpen*)
ACTION ACheckColumns: #BEGIN_EDIT_BLOCK
aIsAnyColumnActive(bActive => bColumnActive);

;#END_EDIT_BLOCK END_ACTION (*ACheckColumns*)
STEP Step24:
END_STEP

STEP S_AfterCycleLoop:
AStepsAfterCycle (P);
ARunStepsAfterCycle (N);
END_STEP

ACTION AStepsAfterCycle: #BEGIN_EDIT_BLOCK
abInterpreter.aInitInterpreter(iColumn := 1,
                               iRow := g_iAutoCycleLoopEndLine,
                               iEndRow := sv_iUsedRows,
                               bSkipAlreadyPosReached := FALSE,
                               bExcludeActiveColumns := FALSE);

abInterpreter.aIncreaseRow(iColumn := 1,
                           iEndRow := sv_iUsedRows);

;#END_EDIT_BLOCK END_ACTION (*AStepsAfterCycle*)
ACTION ARunStepsAfterCycle: #BEGIN_EDIT_BLOCK
abInterpreter.aInterpret();
abInterpreter.aStatus();

;#END_EDIT_BLOCK END_ACTION (*ARunStepsAfterCycle*)
STEP S_WaitReady:
END_STEP

STEP S_End:
Action35 (P);
END_STEP

ACTION Action35: #BEGIN_EDIT_BLOCK
bReady := TRUE;
IF (sv_OperationMode <> nFullAutomatic) THEN
   sv_bAutoCycleRunning := FALSE;
END_IF;
g_SafetyData.MovementToActivate := 0;

;#END_EDIT_BLOCK END_ACTION (*Action35*)

(* transitions *)
GO_ON_TRANSITION T_StartCondOK (* Trans1 *) FROM S_CheckStartCond TO S_CheckStartCycle :=  #BEGIN_EDIT_BLOCK
NOT bStopCycle AND NOT bStopAfterCycle
;#END_EDIT_BLOCK
END_TRANSITION

GO_ON_TRANSITION T_StartCycle (* Trans2 *) FROM S_CheckStartCycle TO Step42 :=  #BEGIN_EDIT_BLOCK
bCanStart AND bDelayExceeded AND NOT mbRecalcActive
;#END_EDIT_BLOCK
END_TRANSITION

GO_ON_TRANSITION TSequenceInterrupted (* Trans48 *) FROM Step42 TO Step43 :=  #BEGIN_EDIT_BLOCK
sv_bSequenceInterruption
;#END_EDIT_BLOCK
END_TRANSITION

TRANSITION TContinueSequence (* Trans50 *) FROM Step43 TO Step20 :=  #BEGIN_EDIT_BLOCK
NOT sv_bSequenceInterruption
;#END_EDIT_BLOCK
END_TRANSITION

TRANSITION Trans51 (* Trans51 *) FROM Step43 TO Step44 :=  #BEGIN_EDIT_BLOCK
di_StepFwd
;#END_EDIT_BLOCK
END_TRANSITION

GO_ON_TRANSITION TMovementsBeforeCycle (* Trans52 *) FROM Step44 TO S_BeforeCycleLoop :=  #BEGIN_EDIT_BLOCK
bMovesBeforeAutoLoop
;#END_EDIT_BLOCK
END_TRANSITION

GO_ON_TRANSITION TNoMoveBeforeAutocycle (* Trans53 *) FROM Step44 TO S_ODC1 :=  #BEGIN_EDIT_BLOCK
NOT bMovesBeforeAutoLoop

;#END_EDIT_BLOCK
END_TRANSITION

GO_ON_TRANSITION Trans49 (* Trans49 *) FROM Step42 TO Step20 :=  #BEGIN_EDIT_BLOCK
NOT sv_bSequenceInterruption
;#END_EDIT_BLOCK
END_TRANSITION

GO_ON_TRANSITION TFirstCycle (* Trans19 *) FROM Step20 TO S_EjectorAutoBwd :=  #BEGIN_EDIT_BLOCK
sv_bFirstCycle
;#END_EDIT_BLOCK
END_TRANSITION

GO_ON_TRANSITION TEjectorStarted (* Trans12 *) FROM S_EjectorAutoBwd TO S_CheckEjectorBwd :=  #BEGIN_EDIT_BLOCK
bEjectorBwdStarted AND pbEjectorReady^
;#END_EDIT_BLOCK
END_TRANSITION

GO_ON_TRANSITION TEjectorBwd (* Trans10 *) FROM S_CheckEjectorBwd TO S_BeforeCycleLoop :=  #BEGIN_EDIT_BLOCK
pbEjectorBwd^
;#END_EDIT_BLOCK
END_TRANSITION

GO_ON_TRANSITION TEjectorNotStarted (* Trans13 *) FROM S_EjectorAutoBwd TO S_BeforeCycleLoop :=  #BEGIN_EDIT_BLOCK
NOT bEjectorBwdStarted
;#END_EDIT_BLOCK
END_TRANSITION

TRANSITION TBeforeCycleReady (* Trans17 *) FROM S_BeforeCycleLoop TO S_ODC1 :=  #BEGIN_EDIT_BLOCK
abInterpreter.aStatus.bFinished
;#END_EDIT_BLOCK
END_TRANSITION

GO_ON_TRANSITION TNotFirstCycle (* Trans42 *) FROM Step20 TO S_ODC1 :=  #BEGIN_EDIT_BLOCK
NOT sv_bFirstCycle
;#END_EDIT_BLOCK
END_TRANSITION

GO_ON_TRANSITION Trans32 (* Trans32 *) FROM S_ODC1 TO S_Run :=  #BEGIN_EDIT_BLOCK
TRUE
;#END_EDIT_BLOCK
END_TRANSITION

GO_ON_TRANSITION T_ODCFinished (* Trans17 *) FROM S_Run TO S_FinishCycle :=  #BEGIN_EDIT_BLOCK
abInterpreter.aStatus.bFinished
;#END_EDIT_BLOCK
END_TRANSITION

GO_ON_TRANSITION T_ODCError (* Trans3 *) FROM S_Run TO SErrorWait :=  #BEGIN_EDIT_BLOCK
abInterpreter.aStatus.bError
;#END_EDIT_BLOCK
END_TRANSITION

TRANSITION TStop (* Trans4 *) FROM SErrorWait TO S_CheckStartCond :=  #BEGIN_EDIT_BLOCK
bStopCycle
;#END_EDIT_BLOCK
END_TRANSITION

TRANSITION Trans52 (* Trans75 *) FROM S_FinishCycle TO S_CheckStopCycle :=  #BEGIN_EDIT_BLOCK
TRUE
;#END_EDIT_BLOCK
(*must be IEC transition because of shot counter / production counter*)
END_TRANSITION

GO_ON_TRANSITION T_NewCycle (* Trans13 *) FROM S_CheckStopCycle TO S_CheckStartCycle :=  #BEGIN_EDIT_BLOCK
NOT bStopAfterCycle AND
NOT bDoRecalc
;#END_EDIT_BLOCK
END_TRANSITION

GO_ON_TRANSITION TStopOrRecalc (* Trans28 *) FROM S_CheckStopCycle TO Step27 :=  #BEGIN_EDIT_BLOCK
bStopAfterCycle OR bDoRecalc
;#END_EDIT_BLOCK
END_TRANSITION

GO_ON_TRANSITION Trans21 (* Trans21 *) FROM Step27 TO S_FinishParallelOpen :=  #BEGIN_EDIT_BLOCK
//"parallel open" movements must also be finished
bColumnActive
;#END_EDIT_BLOCK
END_TRANSITION

TRANSITION Trans23 (* Trans23 *) FROM S_FinishParallelOpen TO Step24 :=  #BEGIN_EDIT_BLOCK
NOT bColumnActive
;#END_EDIT_BLOCK
END_TRANSITION

GO_ON_TRANSITION Trans24 (* Trans24 *) FROM Step24 TO S_AfterCycleLoop :=  #BEGIN_EDIT_BLOCK
bStopAfterCycle
;#END_EDIT_BLOCK
END_TRANSITION

GO_ON_TRANSITION Trans27 (* Trans27 *) FROM Step24 TO S_CheckStartCycle :=  #BEGIN_EDIT_BLOCK
bDoRecalc
;#END_EDIT_BLOCK
END_TRANSITION

GO_ON_TRANSITION Trans22 (* Trans22 *) FROM Step27 TO S_AfterCycleLoop :=  #BEGIN_EDIT_BLOCK
NOT bColumnActive
;#END_EDIT_BLOCK
END_TRANSITION

GO_ON_TRANSITION Trans14 (* Trans14 *) FROM S_AfterCycleLoop TO S_WaitReady :=  #BEGIN_EDIT_BLOCK
abInterpreter.aStatus.bFinished
;#END_EDIT_BLOCK
END_TRANSITION

GO_ON_TRANSITION TAllMovementsReady (* Trans8 *) FROM S_WaitReady TO S_End :=  #BEGIN_EDIT_BLOCK
//wait untill all movements are ready
//for example airvalve movement can be still active
sv_StartedManualMovements.iStartedMovements = 0
;#END_EDIT_BLOCK
END_TRANSITION

TRANSITION Trans15 (* Trans15 *) FROM S_End TO S_CheckStartCycle :=  #BEGIN_EDIT_BLOCK
TRUE
;#END_EDIT_BLOCK
END_TRANSITION

(* end IecGraph-Code *)
(* sfc-code *)

(* stand alone actions *)
ACTION ADelayCycle: #BEGIN_EDIT_BLOCK
(**************************************** WARNING ********************************************
 *** The KEBA Kemro K2 System including software is not intended for safety control tasks! ***
 ***                       For further information see Comment tab!                        ***
 *********************************************************************************************)

//delay should not be executed in first cycle
IF sv_bFirstCycle THEN
   bDelayExceeded := TRUE;
ELSE
   IF sv_dCycleDelaySet > t#0s THEN
      sv_dCycleDelayAct := MIN(S_CheckStartCycle.T, sv_dCycleDelaySet);
   ELSE
      sv_dCycleDelayAct := t#0s;
   END_IF;
   bDelayExceeded := S_CheckStartCycle.T >= sv_dCycleDelaySet;
END_IF;

;#END_EDIT_BLOCK END_ACTION (*ADelayCycle*)
ACTION AEjectorAutoBwd: #BEGIN_EDIT_BLOCK
(**************************************** WARNING ********************************************
 *** The KEBA Kemro K2 System including software is not intended for safety control tasks! ***
 ***                       For further information see Comment tab!                        ***
 *********************************************************************************************)

IF mbEjeBwdAtCycleStart AND NOT pbEjectorBwd^ AND NOT bEjectorBwdStarted THEN
   //only start ejector auto bwd movement if the ejector must be bwd at the beginning of the cycle
   //this information is taken from the safety array of the first step

   //modify pbActivated^ because otherwise the ejector will not move bwd if it is switched off
   sv_MovementsAvailable[iMoveNrEjectorBwd].pMovementData^.pbActivated := @sv_bTRUE;

   //attention:
   //if ejector is not programmed in sequence, there are no safety conditions for ejector bwd movement
   aStartSingleMovement(DeviceId := DeviceIdEjector,
                        MoveDir := cMoveBwd,
                        MoveId := cMoveBwd,
                        bNeedCheckSafety := sv_MovementsAvailable[iMoveNrEjectorBwd].pMovementData^.bProgrammedInSequence);

   bEjectorBwdStarted := TRUE;
END_IF;

;#END_EDIT_BLOCK END_ACTION (*AEjectorAutoBwd*)
ACTION AInitEjectorBwd: #BEGIN_EDIT_BLOCK
(**************************************** WARNING ********************************************
 *** The KEBA Kemro K2 System including software is not intended for safety control tasks! ***
 ***                       For further information see Comment tab!                        ***
 *********************************************************************************************)

IF NOT bInitDone THEN
   fbGetMoveNumber(DeviceId := DeviceIdEjector,
                   MoveId := cMoveBwd,
                   MoveDir := cMoveBwd);

   IF fbGetMoveNumber.bFound THEN
      iMoveNrEjectorBwd := fbGetMoveNumber.iMoveNumber;
      pbEjectorBwd := sv_MovementsAvailable[fbGetMoveNumber.iMoveNumber].pMovementData^.pbPosReached;
      pbEjectorBwdActivated := sv_MovementsAvailable[fbGetMoveNumber.iMoveNumber].pMovementData^.pbActivated;
      pbEjectorReady := sv_MovementsAvailable[fbGetMoveNumber.iMoveNumber].pbDeviceReady;
   ELSE
      //ejector bwd movement not found
      pbEjectorBwd := @sv_bTRUE;
      pbEjectorBwdActivated := @sv_bTRUE;
      pbEjectorReady := @sv_bTRUE;
   END_IF;

   bInitDone := TRUE;
END_IF;

;#END_EDIT_BLOCK END_ACTION (*AInitEjectorBwd*)
ACTION ACheckEjectorBwd: #BEGIN_EDIT_BLOCK
(**************************************** WARNING ********************************************
 *** The KEBA Kemro K2 System including software is not intended for safety control tasks! ***
 ***                       For further information see Comment tab!                        ***
 *********************************************************************************************)

//set pbActivated to original reference
sv_MovementsAvailable[iMoveNrEjectorBwd].pMovementData^.pbActivated := pbEjectorBwdActivated;
bEjectorBwdStarted := FALSE;

IF NOT pbEjectorBwd^ THEN
   //ejector is not bwd -> set according alarm
   SET_ALARM(Name := sv_MovementsAvailable[iMoveNrEjectorBwd].pMovementData^.Alarm.AlarmId,
             SubID1 := sv_MovementsAvailable[iMoveNrEjectorBwd].pMovementData^.Alarm.SubId[1],
             SubID2 := sv_MovementsAvailable[iMoveNrEjectorBwd].pMovementData^.Alarm.SubId[2],
             SubID3 := sv_MovementsAvailable[iMoveNrEjectorBwd].pMovementData^.Alarm.SubId[3],
             SubID4 := sv_MovementsAvailable[iMoveNrEjectorBwd].pMovementData^.Alarm.SubId[4]);

   //switch to manual mode
   fbAutoManual();
END_IF;

;#END_EDIT_BLOCK END_ACTION (*ACheckEjectorBwd*)
ACTION AInitInterpreter: #BEGIN_EDIT_BLOCK
(**************************************** WARNING ********************************************
 *** The KEBA Kemro K2 System including software is not intended for safety control tasks! ***
 ***                       For further information see Comment tab!                        ***
 *********************************************************************************************)

aClearStepState(TRUE);
abInterpreter.aInitInterpreter(iColumn := 1,
                               iRow := g_iAutoCycleLoopStartLine,
                               iEndRow := g_iAutoCycleLoopEndLine,
                               bSkipAlreadyPosReached := FALSE,
                               bExcludeActiveColumns := TRUE);

//find first "valid" line to save cycle time
abInterpreter.aIncreaseRow(iColumn := 1,
                           iEndRow := g_iAutoCycleLoopEndLine);

;#END_EDIT_BLOCK END_ACTION (*AInitInterpreter*)
ACTION AStartCycle: #BEGIN_EDIT_BLOCK
(**************************************** WARNING ********************************************
 *** The KEBA Kemro K2 System including software is not intended for safety control tasks! ***
 ***                       For further information see Comment tab!                        ***
 *********************************************************************************************)

IF NOT sv_bFirstCycle THEN
   //check of cycle time at the beginning of first cycle is not necessary
   aCheckCycleTime();
END_IF;

//save last cycle time
sv_dLastCycleTime := sv_dCycleTime;

mbCycleTimeRunning := TRUE;

//reset timers
mbResetCycleTime := TRUE;
mbResetCycleTimeMachine := TRUE;

sv_bAutoCycleRunning := TRUE;
mbCycleTimeMachineRunning := TRUE;

SET_EVENT(evNewCycleStarted);

;#END_EDIT_BLOCK END_ACTION (*AStartCycle*)

(* exits *)

EXIT_TRANSITION StopAllMoves := #BEGIN_EDIT_BLOCK
bStopCycle
;#END_EDIT_BLOCK
PRIORITY 1 WITH
(* init step *)
INITIAL_STEP S_StopAllMoves:
AStopInterpreter (P);
END_STEP

ACTION AStopInterpreter: #BEGIN_EDIT_BLOCK
abInterpreter.aStopInterpreterNormal();

;#END_EDIT_BLOCK END_ACTION (*AStopInterpreter*)
STEP S_CheckStartCond:
AAutoCycleReady (P);
END_STEP

(* steps *)

(* transitions *)
TRANSITION T_CheckStop (* Trans12 *) FROM S_StopAllMoves TO S_CheckStartCond :=  #BEGIN_EDIT_BLOCK
TRUE
;#END_EDIT_BLOCK
END_TRANSITION
